LIN {X 0,Y 475.19,Z 422.26,A -85,B 0,C 180,E1 -7300.869,E2 -7300.869} C_VEL
LIN {X 0,Y 475.479,Z 413.975,A -85,B 0,C 180,E1 -7301.294,E2 -7301.294} C_VEL
LIN {X 0,Y 475.705,Z 405.069,A -85,B 0,C 180,E1 -7301.64,E2 -7301.64} C_VEL
LIN {X 0,Y 475.915,Z 396.208,A -85,B 0,C 180,E1 -7301.877,E2 -7301.877} C_VEL
LIN {X 0,Y 476.151,Z 333.395,A -85,B 0,C 180,E1 -7302.878,E2 -7302.878} C_VEL
LIN {X 0,Y 474.49,Z 318.296,A -85,B 0,C 180,E1 -7303.182,E2 -7303.182} C_VEL
LIN {X 0,Y 474.879,Z 302.969,A -85,B 0,C 180,E1 -7305.982,E2 -7305.982} C_VEL
LIN {X 0,Y 475.373,Z 286.697,A -85,B 0,C 180,E1 -7308.981,E2 -7308.981} C_VEL
LIN {X 0,Y 476.015,Z 268.666,A -85,B 0,C 180,E1 -7312.345,E2 -7312.345} C_VEL
LIN {X 0,Y 476.027,Z 263.851,A -85,B 0,C 180,E1 -7313.262,E2 -7313.262} C_VEL
LIN {X 0,Y 474.659,Z 256.174,A -85,B 0,C 180,E1 -7314.843,E2 -7314.843} C_VEL
LIN {X 0,Y 474.641,Z 256.171,A -85,B 0,C 180,E1 -7318.282,E2 -7318.282} C_VEL
LIN {X 0,Y 474.599,Z 256.179,A -85,B 0,C 180,E1 -7321.217,E2 -7321.217} C_VEL
LIN {X 0,Y 474.632,Z 256.171,A -85,B 0,C 180,E1 -7324.241,E2 -7324.241} C_VEL
LIN {X 0,Y 474.589,Z 256.182,A -85,B 0,C 180,E1 -7327.383,E2 -7327.383} C_VEL
LIN {X 0,Y 474.626,Z 256.178,A -85,B 0,C 180,E1 -7329.647,E2 -7329.647} C_VEL
LIN {X 0,Y 474.614,Z 256.174,A -85,B 0,C 180,E1 -7332.934,E2 -7332.934} C_VEL
LIN {X 0,Y 474.606,Z 256.177,A -85,B 0,C 180,E1 -7335.894,E2 -7335.894} C_VEL
LIN {X 0,Y 474.626,Z 256.173,A -85,B 0,C 180,E1 -7339.04,E2 -7339.04} C_VEL
LIN {X 0,Y 474.608,Z 256.18,A -85,B 0,C 180,E1 -7341.703,E2 -7341.703} C_VEL
LIN {X 0,Y 474.626,Z 256.172,A -85,B 0,C 180,E1 -7344.725,E2 -7344.725} C_VEL
LIN {X 0,Y 474.632,Z 256.176,A -85,B 0,C 180,E1 -7347.787,E2 -7347.787} C_VEL
LIN {X 0,Y 474.62,Z 256.173,A -85,B 0,C 180,E1 -7350.884,E2 -7350.884} C_VEL
LIN {X 0,Y 474.664,Z 256.174,A -85,B 0,C 180,E1 -7353.628,E2 -7353.628} C_VEL
LIN {X 0,Y 474.632,Z 256.171,A -85,B 0,C 180,E1 -7356.64,E2 -7356.64} C_VEL
LIN {X 0,Y 474.65,Z 256.17,A -85,B 0,C 180,E1 -7360.089,E2 -7360.089} C_VEL
LIN {X 0,Y 474.645,Z 256.169,A -85,B 0,C 180,E1 -7362.774,E2 -7362.774} C_VEL
LIN {X 0,Y 474.643,Z 256.176,A -85,B 0,C 180,E1 -7365.42,E2 -7365.42} C_VEL
LIN {X 0,Y 474.698,Z 256.165,A -85,B 0,C 180,E1 -7368.037,E2 -7368.037} C_VEL
LIN {X 0,Y 474.723,Z 256.167,A -85,B 0,C 180,E1 -7371.486,E2 -7371.486} C_VEL
LIN {X 0,Y 474.773,Z 256.155,A -85,B 0,C 180,E1 -7374.052,E2 -7374.052} C_VEL
LIN {X 0,Y 474.888,Z 256.145,A -85,B 0,C 180,E1 -7377.455,E2 -7377.455} C_VEL
LIN {X 0,Y 474.905,Z 256.139,A -85,B 0,C 180,E1 -7379.999,E2 -7379.999} C_VEL
LIN {X 0,Y 474.888,Z 256.139,A -85,B 0,C 180,E1 -7382.544,E2 -7382.544} C_VEL
LIN {X 0,Y 474.772,Z 256.157,A -85,B 0,C 180,E1 -7385.947,E2 -7385.947} C_VEL
LIN {X 0,Y 474.721,Z 256.16,A -85,B 0,C 180,E1 -7388.513,E2 -7388.513} C_VEL
LIN {X 0,Y 474.731,Z 256.162,A -85,B 0,C 180,E1 -7391.961,E2 -7391.961} C_VEL
LIN {X 0,Y 474.672,Z 256.171,A -85,B 0,C 180,E1 -7395.767,E2 -7395.767} C_VEL
LIN {X 0,Y 474.657,Z 256.169,A -85,B 0,C 180,E1 -7399.01,E2 -7399.01} C_VEL
LIN {X 0,Y 474.581,Z 256.183,A -85,B 0,C 180,E1 -7401.728,E2 -7401.728} C_VEL
LIN {X 0,Y 474.65,Z 256.169,A -85,B 0,C 180,E1 -7404.492,E2 -7404.492} C_VEL
LIN {X 0,Y 474.69,Z 256.168,A -85,B 0,C 180,E1 -7407.338,E2 -7407.338} C_VEL
LIN {X 0,Y 474.596,Z 256.176,A -85,B 0,C 180,E1 -7410.81,E2 -7410.81} C_VEL
LIN {X 0,Y 474.629,Z 256.174,A -85,B 0,C 180,E1 -7413.984,E2 -7413.984} C_VEL
LIN {X 0,Y 474.566,Z 256.18,A -85,B 0,C 180,E1 -7416.9,E2 -7416.9} C_VEL
LIN {X 0,Y 474.643,Z 256.177,A -85,B 0,C 180,E1 -7419.651,E2 -7419.651} C_VEL
LIN {X 0,Y 474.626,Z 256.173,A -85,B 0,C 180,E1 -7422.931,E2 -7422.931} C_VEL
LIN {X 0,Y 474.609,Z 256.178,A -85,B 0,C 180,E1 -7425.896,E2 -7425.896} C_VEL
LIN {X 0,Y 474.636,Z 256.172,A -85,B 0,C 180,E1 -7429.038,E2 -7429.038} C_VEL
LIN {X 0,Y 474.607,Z 256.181,A -85,B 0,C 180,E1 -7431.703,E2 -7431.703} C_VEL
LIN {X 0,Y 474.619,Z 256.173,A -85,B 0,C 180,E1 -7434.726,E2 -7434.726} C_VEL
LIN {X 0,Y 474.628,Z 256.177,A -85,B 0,C 180,E1 -7437.788,E2 -7437.788} C_VEL
LIN {X 0,Y 474.614,Z 256.174,A -85,B 0,C 180,E1 -7440.884,E2 -7440.884} C_VEL
LIN {X 0,Y 474.652,Z 256.177,A -85,B 0,C 180,E1 -7443.628,E2 -7443.628} C_VEL
LIN {X 0,Y 474.627,Z 256.172,A -85,B 0,C 180,E1 -7446.641,E2 -7446.641} C_VEL
LIN {X 0,Y 474.648,Z 256.171,A -85,B 0,C 180,E1 -7450.089,E2 -7450.089} C_VEL
LIN {X 0,Y 474.646,Z 256.173,A -85,B 0,C 180,E1 -7451.682,E2 -7451.682} C_VEL
LIN {X 0,Y 473.984,Z 256.257,A -85,B 0,C 180,E1 -7452.391,E2 -7452.391} C_VEL
LIN {X 0,Y 471.132,Z 256.614,A -85,B 0,C 180,E1 -7453.542,E2 -7453.542} C_VEL
LIN {X 0,Y 468.716,Z 256.913,A -85,B 0,C 180,E1 -7454.47,E2 -7454.47} C_VEL
LIN {X 0,Y 467.674,Z 257.041,A -85,B 0,C 180,E1 -7455.188,E2 -7455.188} C_VEL
LIN {X 0,Y 467.587,Z 257.05,A -85,B 0,C 180,E1 -7455.431,E2 -7455.431} C_VEL
LIN {X 0,Y 467.646,Z 257.042,A -85,B 0,C 180,E1 -7458.734,E2 -7458.734} C_VEL
LIN {X 0,Y 467.74,Z 257.031,A -85,B 0,C 180,E1 -7462.228,E2 -7462.228} C_VEL
LIN {X 0,Y 467.711,Z 257.034,A -85,B 0,C 180,E1 -7464.827,E2 -7464.827} C_VEL
LIN {X 0,Y 467.849,Z 257.021,A -85,B 0,C 180,E1 -7467.417,E2 -7467.417} C_VEL
LIN {X 0,Y 467.871,Z 257.017,A -85,B 0,C 180,E1 -7470,E2 -7470} C_VEL
LIN {X 0,Y 467.849,Z 257.017,A -85,B 0,C 180,E1 -7472.583,E2 -7472.583} C_VEL
LIN {X 0,Y 467.722,Z 257.035,A -85,B 0,C 180,E1 -7476.037,E2 -7476.037} C_VEL
LIN {X 0,Y 467.671,Z 257.039,A -85,B 0,C 180,E1 -7478.643,E2 -7478.643} C_VEL
LIN {X 0,Y 467.673,Z 257.04,A -85,B 0,C 180,E1 -7482.145,E2 -7482.145} C_VEL
LIN {X 0,Y 467.639,Z 257.047,A -85,B 0,C 180,E1 -7485.885,E2 -7485.885} C_VEL
LIN {X 0,Y 467.612,Z 257.049,A -85,B 0,C 180,E1 -7489.308,E2 -7489.308} C_VEL
LIN {X 0,Y 467.523,Z 257.06,A -85,B 0,C 180,E1 -7492.074,E2 -7492.074} C_VEL
LIN {X 0,Y 467.567,Z 257.053,A -85,B 0,C 180,E1 -7494.889,E2 -7494.889} C_VEL
LIN {X 0,Y 467.604,Z 257.053,A -85,B 0,C 180,E1 -7497.769,E2 -7497.769} C_VEL
LIN {X 0,Y 467.536,Z 257.057,A -85,B 0,C 180,E1 -7501.041,E2 -7501.041} C_VEL
LIN {X 0,Y 467.613,Z 257.233,A -85,B 0,C 180,E1 -7502.883,E2 -7502.883} C_VEL
LIN {X 0,Y 467.517,Z 268.713,A -85,B 0,C 180,E1 -7505.711,E2 -7505.711} C_VEL
LIN {X 0,Y 469.565,Z 280.34,A -85,B 0,C 180,E1 -7505.973,E2 -7505.973} C_VEL
LIN {X 0,Y 469.055,Z 344.667,A -85,B 0,C 180,E1 -7507.011,E2 -7507.011} C_VEL
LIN {X 0,Y 468.902,Z 354.626,A -85,B 0,C 180,E1 -7507.29,E2 -7507.29} C_VEL
LIN {X 0,Y 468.743,Z 365.834,A -85,B 0,C 180,E1 -7507.764,E2 -7507.764} C_VEL
LIN {X 0,Y 468.444,Z 375.752,A -85,B 0,C 180,E1 -7508.357,E2 -7508.357} C_VEL
LIN {X 0,Y 468.184,Z 385.112,A -85,B 0,C 180,E1 -7509.084,E2 -7509.084} C_VEL
LIN {X 0,Y 467.91,Z 392.862,A -85,B 0,C 180,E1 -7509.83,E2 -7509.83} C_VEL
LIN {X 0,Y 467.618,Z 400.12,A -85,B 0,C 180,E1 -7510.684,E2 -7510.684} C_VEL
LIN {X 0,Y 467.375,Z 407.099,A -85,B 0,C 180,E1 -7511.691,E2 -7511.691} C_VEL
LIN {X 0,Y 467.151,Z 413.62,A -85,B 0,C 180,E1 -7512.888,E2 -7512.888} C_VEL
LIN {X 0,Y 466.987,Z 418.643,A -85,B 0,C 180,E1 -7514.098,E2 -7514.098} C_VEL
LIN {X 0,Y 466.865,Z 421.688,A -85,B 0,C 180,E1 -7515.032,E2 -7515.032} C_VEL
LIN {X 0,Y 466.759,Z 424.644,A -85,B 0,C 180,E1 -7516.279,E2 -7516.279} C_VEL
LIN {X 0,Y 466.656,Z 426.538,A -85,B 0,C 180,E1 -7517.556,E2 -7517.556} C_VEL
LIN {X 0,Y 466.634,Z 427.345,A -85,B 0,C 180,E1 -7518.854,E2 -7518.854} C_VEL
LIN {X 0,Y 466.617,Z 426.997,A -85,B 0,C 180,E1 -7520.186,E2 -7520.186} C_VEL
LIN {X 0,Y 466.747,Z 424.688,A -85,B 0,C 180,E1 -7521.878,E2 -7521.878} C_VEL
LIN {X 0,Y 466.892,Z 422.133,A -85,B 0,C 180,E1 -7522.98,E2 -7522.98} C_VEL
LIN {X 0,Y 467.045,Z 417.704,A -85,B 0,C 180,E1 -7524.347,E2 -7524.347} C_VEL
LIN {X 0,Y 467.258,Z 412.531,A -85,B 0,C 180,E1 -7525.507,E2 -7525.507} C_VEL
LIN {X 0,Y 467.451,Z 407.21,A -85,B 0,C 180,E1 -7526.461,E2 -7526.461} C_VEL
LIN {X 0,Y 467.698,Z 399.703,A -85,B 0,C 180,E1 -7527.537,E2 -7527.537} C_VEL
LIN {X 0,Y 468.021,Z 393.235,A -85,B 0,C 180,E1 -7528.294,E2 -7528.294} C_VEL
LIN {X 0,Y 468.283,Z 385.422,A -85,B 0,C 180,E1 -7529.052,E2 -7529.052} C_VEL
LIN {X 0,Y 468.555,Z 376.993,A -85,B 0,C 180,E1 -7529.713,E2 -7529.713} C_VEL
LIN {X 0,Y 468.813,Z 365.724,A -85,B 0,C 180,E1 -7530.396,E2 -7530.396} C_VEL
LIN {X 0,Y 469.014,Z 354.621,A -85,B 0,C 180,E1 -7530.858,E2 -7530.858} C_VEL
LIN {X 0,Y 469.141,Z 345.648,A -85,B 0,C 180,E1 -7531.112,E2 -7531.112} C_VEL
LIN {X 0,Y 469.662,Z 279.9,A -85,B 0,C 180,E1 -7532.183,E2 -7532.183} C_VEL
LIN {X 0,Y 467.626,Z 268.438,A -85,B 0,C 180,E1 -7532.461,E2 -7532.461} C_VEL
LIN {X 0,Y 467.522,Z 257.064,A -85,B 0,C 180,E1 -7534.853,E2 -7534.853} C_VEL
LIN {X 0,Y 467.559,Z 257.059,A -85,B 0,C 180,E1 -7536.996,E2 -7536.996} C_VEL
LIN {X 0,Y 467.612,Z 257.051,A -85,B 0,C 180,E1 -7539.778,E2 -7539.778} C_VEL
LIN {X 0,Y 467.598,Z 257.056,A -85,B 0,C 180,E1 -7542.507,E2 -7542.507} C_VEL
LIN {X 0,Y 467.595,Z 257.05,A -85,B 0,C 180,E1 -7545.197,E2 -7545.197} C_VEL
LIN {X 0,Y 467.646,Z 257.043,A -85,B 0,C 180,E1 -7547.855,E2 -7547.855} C_VEL
LIN {X 0,Y 467.672,Z 257.04,A -85,B 0,C 180,E1 -7551.358,E2 -7551.358} C_VEL
LIN {X 0,Y 467.737,Z 257.033,A -85,B 0,C 180,E1 -7553.963,E2 -7553.963} C_VEL
LIN {X 0,Y 467.851,Z 257.014,A -85,B 0,C 180,E1 -7557.418,E2 -7557.418} C_VEL
LIN {X 0,Y 467.872,Z 257.016,A -85,B 0,C 180,E1 -7560.001,E2 -7560.001} C_VEL
LIN {X 0,Y 467.851,Z 257.023,A -85,B 0,C 180,E1 -7562.584,E2 -7562.584} C_VEL
LIN {X 0,Y 467.735,Z 257.032,A -85,B 0,C 180,E1 -7566.038,E2 -7566.038} C_VEL
LIN {X 0,Y 467.673,Z 257.042,A -85,B 0,C 180,E1 -7568.644,E2 -7568.644} C_VEL
LIN {X 0,Y 467.647,Z 257.044,A -85,B 0,C 180,E1 -7572.146,E2 -7572.146} C_VEL
LIN {X 0,Y 467.631,Z 257.043,A -85,B 0,C 180,E1 -7575.696,E2 -7575.696} C_VEL
LIN {X 0,Y 467.61,Z 257.05,A -85,B 0,C 180,E1 -7578.766,E2 -7578.766} C_VEL
LIN {X 0,Y 467.573,Z 257.047,A -85,B 0,C 180,E1 -7581.269,E2 -7581.269} C_VEL
LIN {X 0,Y 467.566,Z 257.052,A -85,B 0,C 180,E1 -7583.944,E2 -7583.944} C_VEL
LIN {X 0,Y 467.622,Z 257.049,A -85,B 0,C 180,E1 -7586.8,E2 -7586.8} C_VEL
LIN {X 0,Y 467.581,Z 257.045,A -85,B 0,C 180,E1 -7589.737,E2 -7589.737} C_VEL
LIN {X 0,Y 467.578,Z 257.05,A -85,B 0,C 180,E1 -7592.759,E2 -7592.759} C_VEL
LIN {X 0,Y 467.552,Z 257.055,A -85,B 0,C 180,E1 -7595.89,E2 -7595.89} C_VEL
LIN {X 0,Y 467.61,Z 257.047,A -85,B 0,C 180,E1 -7599.142,E2 -7599.142} C_VEL
LIN {X 0,Y 467.582,Z 257.056,A -85,B 0,C 180,E1 -7602.568,E2 -7602.568} C_VEL
LIN {X 0,Y 467.566,Z 257.054,A -85,B 0,C 180,E1 -7605.054,E2 -7605.054} C_VEL
LIN {X 0,Y 467.586,Z 257.049,A -85,B 0,C 180,E1 -7607.441,E2 -7607.441} C_VEL
LIN {X 0,Y 467.579,Z 257.054,A -85,B 0,C 180,E1 -7610.856,E2 -7610.856} C_VEL
LIN {X 0,Y 467.56,Z 257.058,A -85,B 0,C 180,E1 -7614.261,E2 -7614.261} C_VEL
LIN {X 0,Y 467.58,Z 257.051,A -85,B 0,C 180,E1 -7617.322,E2 -7617.322} C_VEL
LIN {X 0,Y 467.567,Z 257.06,A -85,B 0,C 180,E1 -7620.669,E2 -7620.669} C_VEL
LIN {X 0,Y 467.611,Z 257.049,A -85,B 0,C 180,E1 -7623.2,E2 -7623.2} C_VEL
LIN {X 0,Y 467.641,Z 257.128,A -85,B 0,C 180,E1 -7625.648,E2 -7625.648} C_VEL
LIN {X 0,Y 468.758,Z 264.468,A -85,B 0,C 180,E1 -7627.058,E2 -7627.058} C_VEL
LIN {X 0,Y 468.382,Z 277.023,A -85,B 0,C 180,E1 -7629.353,E2 -7629.353} C_VEL
LIN {X 0,Y 467.915,Z 294.514,A -85,B 0,C 180,E1 -7632.519,E2 -7632.519} C_VEL
LIN {X 0,Y 467.473,Z 314.296,A -85,B 0,C 180,E1 -7636.082,E2 -7636.082} C_VEL
LIN {X 0,Y 467.397,Z 317.179,A -85,B 0,C 180,E1 -7636.592,E2 -7636.592} C_VEL
LIN {X 0,Y 469.438,Z 337,A -85,B 0,C 180,E1 -7636.974,E2 -7636.974} C_VEL
LIN {X 0,Y 469.007,Z 395.268,A -85,B 0,C 180,E1 -7637.918,E2 -7637.918} C_VEL
LIN {X 0,Y 468.757,Z 404.976,A -85,B 0,C 180,E1 -7638.186,E2 -7638.186} C_VEL
LIN {X 0,Y 468.411,Z 416.086,A -85,B 0,C 180,E1 -7638.643,E2 -7638.643} C_VEL
LIN {X 0,Y 468.077,Z 426.991,A -85,B 0,C 180,E1 -7639.292,E2 -7639.292} C_VEL
LIN {X 0,Y 467.789,Z 435.462,A -85,B 0,C 180,E1 -7639.942,E2 -7639.942} C_VEL
LIN {X 0,Y 467.48,Z 443.473,A -85,B 0,C 180,E1 -7640.7,E2 -7640.7} C_VEL
LIN {X 0,Y 467.218,Z 450.966,A -85,B 0,C 180,E1 -7641.567,E2 -7641.567} C_VEL
LIN {X 0,Y 467.042,Z 458.58,A -85,B 0,C 180,E1 -7642.652,E2 -7642.652} C_VEL
LIN {X 0,Y 466.811,Z 465.545,A -85,B 0,C 180,E1 -7643.951,E2 -7643.951} C_VEL
LIN {X 0,Y 466.796,Z 469.281,A -85,B 0,C 180,E1 -7644.817,E2 -7644.817} C_VEL
LIN {X 0,Y 466.686,Z 472.339,A -85,B 0,C 180,E1 -7645.682,E2 -7645.682} C_VEL
LIN {X 0,Y 466.762,Z 474.725,A -85,B 0,C 180,E1 -7646.547,E2 -7646.547} C_VEL
LIN {X 0,Y 466.706,Z 476.52,A -85,B 0,C 180,E1 -7647.411,E2 -7647.411} C_VEL
LIN {X 0,Y 466.693,Z 477.808,A -85,B 0,C 180,E1 -7648.274,E2 -7648.274} C_VEL
LIN {X 0,Y 466.626,Z 478.608,A -85,B 0,C 180,E1 -7649.137,E2 -7649.137} C_VEL
LIN {X 0,Y 466.612,Z 478.919,A -85,B 0,C 180,E1 -7650,E2 -7650} C_VEL
LIN {X 0,Y 466.626,Z 478.632,A -85,B 0,C 180,E1 -7650.863,E2 -7650.863} C_VEL
LIN {X 0,Y 466.693,Z 477.841,A -85,B 0,C 180,E1 -7651.726,E2 -7651.726} C_VEL
LIN {X 0,Y 466.706,Z 476.562,A -85,B 0,C 180,E1 -7652.589,E2 -7652.589} C_VEL
LIN {X 0,Y 466.733,Z 473.612,A -85,B 0,C 180,E1 -7653.885,E2 -7653.885} C_VEL
LIN {X 0,Y 466.722,Z 470.906,A -85,B 0,C 180,E1 -7654.751,E2 -7654.751} C_VEL
LIN {X 0,Y 466.817,Z 467.576,A -85,B 0,C 180,E1 -7655.616,E2 -7655.616} C_VEL
LIN {X 0,Y 466.93,Z 462.172,A -85,B 0,C 180,E1 -7656.73,E2 -7656.73} C_VEL
LIN {X 0,Y 467.067,Z 455.786,A -85,B 0,C 180,E1 -7657.783,E2 -7657.783} C_VEL
LIN {X 0,Y 467.385,Z 447.59,A -85,B 0,C 180,E1 -7658.866,E2 -7658.866} C_VEL
LIN {X 0,Y 467.739,Z 437.953,A -85,B 0,C 180,E1 -7659.841,E2 -7659.841} C_VEL
LIN {X 0,Y 467.979,Z 429.95,A -85,B 0,C 180,E1 -7660.492,E2 -7660.492} C_VEL
LIN {X 0,Y 468.214,Z 421.697,A -85,B 0,C 180,E1 -7661.033,E2 -7661.033} C_VEL
LIN {X 0,Y 468.492,Z 413.353,A -85,B 0,C 180,E1 -7661.465,E2 -7661.465} C_VEL
LIN {X 0,Y 468.773,Z 404.358,A -85,B 0,C 180,E1 -7661.814,E2 -7661.814} C_VEL
LIN {X 0,Y 468.94,Z 395.308,A -85,B 0,C 180,E1 -7662.057,E2 -7662.057} C_VEL
LIN {X 0,Y 469.252,Z 334.358,A -85,B 0,C 180,E1 -7663.041,E2 -7663.041} C_VEL
LIN {X 0,Y 467.423,Z 318.062,A -85,B 0,C 180,E1 -7663.355,E2 -7663.355} C_VEL
LIN {X 0,Y 467.868,Z 302.732,A -85,B 0,C 180,E1 -7666.199,E2 -7666.199} C_VEL
LIN {X 0,Y 468.443,Z 285.102,A -85,B 0,C 180,E1 -7669.5,E2 -7669.5} C_VEL
LIN {X 0,Y 469.163,Z 267.094,A -85,B 0,C 180,E1 -7672.922,E2 -7672.922} C_VEL
LIN {X 0,Y 468.122,Z 259.793,A -85,B 0,C 180,E1 -7674.384,E2 -7674.384} C_VEL
LIN {X 0,Y 467.613,Z 257.052,A -85,B 0,C 180,E1 -7674.992,E2 -7674.992} C_VEL
LIN {X 0,Y 467.616,Z 257.051,A -85,B 0,C 180,E1 -7677.769,E2 -7677.769} C_VEL
LIN {X 0,Y 467.568,Z 257.053,A -85,B 0,C 180,E1 -7681.044,E2 -7681.044} C_VEL
LIN {X 0,Y 467.588,Z 257.048,A -85,B 0,C 180,E1 -7684.242,E2 -7684.242} C_VEL
LIN {X 0,Y 467.547,Z 257.057,A -85,B 0,C 180,E1 -7687.186,E2 -7687.186} C_VEL
LIN {X 0,Y 467.576,Z 257.05,A -85,B 0,C 180,E1 -7690.264,E2 -7690.264} C_VEL
LIN {X 0,Y 467.585,Z 257.048,A -85,B 0,C 180,E1 -7692.566,E2 -7692.566} C_VEL
LIN {X 0,Y 467.569,Z 257.053,A -85,B 0,C 180,E1 -7695.052,E2 -7695.052} C_VEL
LIN {X 0,Y 467.587,Z 257.055,A -85,B 0,C 180,E1 -7697.439,E2 -7697.439} C_VEL
LIN {X 0,Y 467.558,Z 257.053,A -85,B 0,C 180,E1 -7700.852,E2 -7700.852} C_VEL
LIN {X 0,Y 467.56,Z 257.052,A -85,B 0,C 180,E1 -7704.26,E2 -7704.26} C_VEL
LIN {X 0,Y 467.579,Z 257.054,A -85,B 0,C 180,E1 -7707.32,E2 -7707.32} C_VEL
LIN {X 0,Y 467.566,Z 257.051,A -85,B 0,C 180,E1 -7710.667,E2 -7710.667} C_VEL
LIN {X 0,Y 467.625,Z 257.047,A -85,B 0,C 180,E1 -7713.2,E2 -7713.2} C_VEL
LIN {X 0,Y 467.589,Z 257.048,A -85,B 0,C 180,E1 -7716.467,E2 -7716.467} C_VEL
LIN {X 0,Y 467.618,Z 257.05,A -85,B 0,C 180,E1 -7719.776,E2 -7719.776} C_VEL
LIN {X 0,Y 467.604,Z 257.046,A -85,B 0,C 180,E1 -7722.506,E2 -7722.506} C_VEL
LIN {X 0,Y 467.601,Z 257.05,A -85,B 0,C 180,E1 -7725.196,E2 -7725.196} C_VEL
LIN {X 0,Y 467.65,Z 257.045,A -85,B 0,C 180,E1 -7727.854,E2 -7727.854} C_VEL
LIN {X 0,Y 467.676,Z 257.042,A -85,B 0,C 180,E1 -7731.357,E2 -7731.357} C_VEL
LIN {X 0,Y 467.737,Z 257.033,A -85,B 0,C 180,E1 -7733.962,E2 -7733.962} C_VEL
LIN {X 0,Y 467.853,Z 257.021,A -85,B 0,C 180,E1 -7737.416,E2 -7737.416} C_VEL
LIN {X 0,Y 467.876,Z 257.015,A -85,B 0,C 180,E1 -7739.999,E2 -7739.999} C_VEL
LIN {X 0,Y 467.854,Z 257.015,A -85,B 0,C 180,E1 -7742.582,E2 -7742.582} C_VEL
LIN {X 0,Y 467.736,Z 257.032,A -85,B 0,C 180,E1 -7746.037,E2 -7746.037} C_VEL
LIN {X 0,Y 467.674,Z 257.038,A -85,B 0,C 180,E1 -7748.642,E2 -7748.642} C_VEL
LIN {X 0,Y 467.675,Z 257.039,A -85,B 0,C 180,E1 -7752.144,E2 -7752.144} C_VEL
LIN {X 0,Y 467.641,Z 257.046,A -85,B 0,C 180,E1 -7755.885,E2 -7755.885} C_VEL
LIN {X 0,Y 467.616,Z 257.049,A -85,B 0,C 180,E1 -7759.307,E2 -7759.307} C_VEL
LIN {X 0,Y 467.526,Z 257.058,A -85,B 0,C 180,E1 -7762.073,E2 -7762.073} C_VEL
LIN {X 0,Y 467.595,Z 257.049,A -85,B 0,C 180,E1 -7764.887,E2 -7764.887} C_VEL
LIN {X 0,Y 467.618,Z 257.05,A -85,B 0,C 180,E1 -7767.768,E2 -7767.768} C_VEL
LIN {X 0,Y 467.56,Z 257.054,A -85,B 0,C 180,E1 -7771.045,E2 -7771.045} C_VEL
LIN {X 0,Y 467.581,Z 257.05,A -85,B 0,C 180,E1 -7774.242,E2 -7774.242} C_VEL
LIN {X 0,Y 467.542,Z 257.057,A -85,B 0,C 180,E1 -7777.187,E2 -7777.187} C_VEL
LIN {X 0,Y 467.587,Z 257.05,A -85,B 0,C 180,E1 -7780.262,E2 -7780.262} C_VEL
LIN {X 0,Y 467.577,Z 257.05,A -85,B 0,C 180,E1 -7782.567,E2 -7782.567} C_VEL
LIN {X 0,Y 467.561,Z 257.054,A -85,B 0,C 180,E1 -7785.053,E2 -7785.053} C_VEL
LIN {X 0,Y 467.615,Z 257.051,A -85,B 0,C 180,E1 -7787.444,E2 -7787.444} C_VEL
LIN {X 0,Y 467.59,Z 257.049,A -85,B 0,C 180,E1 -7790.857,E2 -7790.857} C_VEL
LIN {X 0,Y 467.553,Z 257.054,A -85,B 0,C 180,E1 -7794.26,E2 -7794.26} C_VEL
LIN {X 0,Y 467.573,Z 257.054,A -85,B 0,C 180,E1 -7797.32,E2 -7797.32} C_VEL
LIN {X 0,Y 467.56,Z 257.052,A -85,B 0,C 180,E1 -7800.667,E2 -7800.667} C_VEL
LIN {X 0,Y 467.607,Z 257.049,A -85,B 0,C 180,E1 -7803.2,E2 -7803.2} C_VEL
LIN {X 0,Y 467.585,Z 257.049,A -85,B 0,C 180,E1 -7806.468,E2 -7806.468} C_VEL
LIN {X 0,Y 467.615,Z 257.051,A -85,B 0,C 180,E1 -7809.777,E2 -7809.777} C_VEL
LIN {X 0,Y 467.6,Z 257.047,A -85,B 0,C 180,E1 -7812.507,E2 -7812.507} C_VEL
LIN {X 0,Y 467.587,Z 257.05,A -85,B 0,C 180,E1 -7815.431,E2 -7815.431} C_VEL
LIN {X 0,Y 466.918,Z 257.135,A -85,B 0,C 180,E1 -7816.15,E2 -7816.15} C_VEL
LIN {X 0,Y 464.075,Z 257.49,A -85,B 0,C 180,E1 -7817.318,E2 -7817.318} C_VEL
LIN {X 0,Y 461.677,Z 257.786,A -85,B 0,C 180,E1 -7818.26,E2 -7818.26} C_VEL
LIN {X 0,Y 460.652,Z 257.914,A -85,B 0,C 180,E1 -7818.988,E2 -7818.988} C_VEL
LIN {X 0,Y 460.57,Z 257.925,A -85,B 0,C 180,E1 -7819.234,E2 -7819.234} C_VEL
LIN {X 0,Y 460.706,Z 257.906,A -85,B 0,C 180,E1 -7822.543,E2 -7822.543} C_VEL
LIN {X 0,Y 460.684,Z 257.909,A -85,B 0,C 180,E1 -7824.748,E2 -7824.748} C_VEL
LIN {X 0,Y 460.79,Z 257.9,A -85,B 0,C 180,E1 -7827.377,E2 -7827.377} C_VEL
LIN {X 0,Y 460.842,Z 257.892,A -85,B 0,C 180,E1 -7830,E2 -7830} C_VEL
LIN {X 0,Y 460.79,Z 257.896,A -85,B 0,C 180,E1 -7832.622,E2 -7832.622} C_VEL
LIN {X 0,Y 460.688,Z 257.91,A -85,B 0,C 180,E1 -7836.13,E2 -7836.13} C_VEL
LIN {X 0,Y 460.618,Z 257.918,A -85,B 0,C 180,E1 -7838.776,E2 -7838.776} C_VEL
LIN {X 0,Y 460.624,Z 257.917,A -85,B 0,C 180,E1 -7842.457,E2 -7842.457} C_VEL
LIN {X 0,Y 460.59,Z 257.924,A -85,B 0,C 180,E1 -7845.997,E2 -7845.997} C_VEL
LIN {X 0,Y 460.559,Z 257.926,A -85,B 0,C 180,E1 -7848.901,E2 -7848.901} C_VEL
LIN {X 0,Y 460.505,Z 257.936,A -85,B 0,C 180,E1 -7851.485,E2 -7851.485} C_VEL
LIN {X 0,Y 460.514,Z 257.931,A -85,B 0,C 180,E1 -7854.333,E2 -7854.333} C_VEL
LIN {X 0,Y 460.566,Z 257.93,A -85,B 0,C 180,E1 -7857.745,E2 -7857.745} C_VEL
LIN {X 0,Y 460.509,Z 257.935,A -85,B 0,C 180,E1 -7861.257,E2 -7861.257} C_VEL
LIN {X 0,Y 460.566,Z 258.083,A -85,B 0,C 180,E1 -7862.799,E2 -7862.799} C_VEL
LIN {X 0,Y 460.508,Z 266.701,A -85,B 0,C 180,E1 -7864.942,E2 -7864.942} C_VEL
LIN {X 0,Y 460.502,Z 269.068,A -85,B 0,C 180,E1 -7865.523,E2 -7865.523} C_VEL
LIN {X 0,Y 462.634,Z 281.728,A -85,B 0,C 180,E1 -7865.802,E2 -7865.802} C_VEL
LIN {X 0,Y 462.115,Z 344.743,A -85,B 0,C 180,E1 -7866.836,E2 -7866.836} C_VEL
LIN {X 0,Y 461.916,Z 354.557,A -85,B 0,C 180,E1 -7867.11,E2 -7867.11} C_VEL
LIN {X 0,Y 461.792,Z 365.886,A -85,B 0,C 180,E1 -7867.59,E2 -7867.59} C_VEL
LIN {X 0,Y 461.491,Z 374.985,A -85,B 0,C 180,E1 -7868.125,E2 -7868.125} C_VEL
LIN {X 0,Y 461.256,Z 384.108,A -85,B 0,C 180,E1 -7868.823,E2 -7868.823} C_VEL
LIN {X 0,Y 460.951,Z 392.262,A -85,B 0,C 180,E1 -7869.599,E2 -7869.599} C_VEL
LIN {X 0,Y 460.635,Z 399.359,A -85,B 0,C 180,E1 -7870.423,E2 -7870.423} C_VEL
LIN {X 0,Y 460.423,Z 405.561,A -85,B 0,C 180,E1 -7871.296,E2 -7871.296} C_VEL
LIN {X 0,Y 460.206,Z 410.973,A -85,B 0,C 180,E1 -7872.216,E2 -7872.216} C_VEL
LIN {X 0,Y 459.977,Z 416.757,A -85,B 0,C 180,E1 -7873.436,E2 -7873.436} C_VEL
LIN {X 0,Y 459.844,Z 421.216,A -85,B 0,C 180,E1 -7874.67,E2 -7874.67} C_VEL
LIN {X 0,Y 459.714,Z 424.44,A -85,B 0,C 180,E1 -7875.931,E2 -7875.931} C_VEL
LIN {X 0,Y 459.591,Z 426.566,A -85,B 0,C 180,E1 -7877.222,E2 -7877.222} C_VEL
LIN {X 0,Y 459.545,Z 427.609,A -85,B 0,C 180,E1 -7878.535,E2 -7878.535} C_VEL
LIN {X 0,Y 459.544,Z 427.488,A -85,B 0,C 180,E1 -7880.036,E2 -7880.036} C_VEL
LIN {X 0,Y 459.618,Z 426.287,A -85,B 0,C 180,E1 -7881.244,E2 -7881.244} C_VEL
LIN {X 0,Y 459.783,Z 423.596,A -85,B 0,C 180,E1 -7882.639,E2 -7882.639} C_VEL
LIN {X 0,Y 459.908,Z 420.353,A -85,B 0,C 180,E1 -7883.782,E2 -7883.782} C_VEL
LIN {X 0,Y 460.073,Z 416.641,A -85,B 0,C 180,E1 -7884.785,E2 -7884.785} C_VEL
LIN {X 0,Y 460.272,Z 411.584,A -85,B 0,C 180,E1 -7885.866,E2 -7885.866} C_VEL
LIN {X 0,Y 460.444,Z 407.035,A -85,B 0,C 180,E1 -7886.669,E2 -7886.669} C_VEL
LIN {X 0,Y 460.666,Z 400.932,A -85,B 0,C 180,E1 -7887.565,E2 -7887.565} C_VEL
LIN {X 0,Y 461.032,Z 393.607,A -85,B 0,C 180,E1 -7888.443,E2 -7888.443} C_VEL
LIN {X 0,Y 461.309,Z 386.075,A -85,B 0,C 180,E1 -7889.186,E2 -7889.186} C_VEL
LIN {X 0,Y 461.596,Z 377.93,A -85,B 0,C 180,E1 -7889.84,E2 -7889.84} C_VEL
LIN {X 0,Y 461.798,Z 368.787,A -85,B 0,C 180,E1 -7890.425,E2 -7890.425} C_VEL
LIN {X 0,Y 462.064,Z 356.373,A -85,B 0,C 180,E1 -7890.996,E2 -7890.996} C_VEL
LIN {X 0,Y 462.219,Z 346.142,A -85,B 0,C 180,E1 -7891.297,E2 -7891.297} C_VEL
LIN {X 0,Y 462.712,Z 280.086,A -85,B 0,C 180,E1 -7892.401,E2 -7892.401} C_VEL
LIN {X 0,Y 460.64,Z 268.889,A -85,B 0,C 180,E1 -7892.666,E2 -7892.666} C_VEL
LIN {X 0,Y 460.634,Z 259.161,A -85,B 0,C 180,E1 -7894.711,E2 -7894.711} C_VEL
LIN {X 0,Y 460.488,Z 257.939,A -85,B 0,C 180,E1 -7895.004,E2 -7895.004} C_VEL
LIN {X 0,Y 460.495,Z 257.937,A -85,B 0,C 180,E1 -7897.572,E2 -7897.572} C_VEL
LIN {X 0,Y 460.558,Z 257.935,A -85,B 0,C 180,E1 -7900.385,E2 -7900.385} C_VEL
LIN {X 0,Y 460.555,Z 257.928,A -85,B 0,C 180,E1 -7903.147,E2 -7903.147} C_VEL
LIN {X 0,Y 460.543,Z 257.929,A -85,B 0,C 180,E1 -7905.868,E2 -7905.868} C_VEL
LIN {X 0,Y 460.603,Z 257.927,A -85,B 0,C 180,E1 -7908.56,E2 -7908.56} C_VEL
LIN {X 0,Y 460.685,Z 257.913,A -85,B 0,C 180,E1 -7912.109,E2 -7912.109} C_VEL
LIN {X 0,Y 460.692,Z 257.912,A -85,B 0,C 180,E1 -7914.749,E2 -7914.749} C_VEL
LIN {X 0,Y 460.816,Z 257.891,A -85,B 0,C 180,E1 -7917.378,E2 -7917.378} C_VEL
LIN {X 0,Y 460.843,Z 257.892,A -85,B 0,C 180,E1 -7920.001,E2 -7920.001} C_VEL
LIN {X 0,Y 460.816,Z 257.898,A -85,B 0,C 180,E1 -7922.623,E2 -7922.623} C_VEL
LIN {X 0,Y 460.701,Z 257.909,A -85,B 0,C 180,E1 -7926.131,E2 -7926.131} C_VEL
LIN {X 0,Y 460.62,Z 257.92,A -85,B 0,C 180,E1 -7928.777,E2 -7928.777} C_VEL
LIN {X 0,Y 460.605,Z 257.921,A -85,B 0,C 180,E1 -7932.446,E2 -7932.446} C_VEL
LIN {X 0,Y 460.592,Z 257.921,A -85,B 0,C 180,E1 -7935.998,E2 -7935.998} C_VEL
LIN {X 0,Y 460.563,Z 257.926,A -85,B 0,C 180,E1 -7938.903,E2 -7938.903} C_VEL
LIN {X 0,Y 460.509,Z 257.927,A -85,B 0,C 180,E1 -7941.487,E2 -7941.487} C_VEL
LIN {X 0,Y 460.536,Z 257.932,A -85,B 0,C 180,E1 -7944.333,E2 -7944.333} C_VEL
LIN {X 0,Y 460.578,Z 257.922,A -85,B 0,C 180,E1 -7947.244,E2 -7947.244} C_VEL
LIN {X 0,Y 460.521,Z 257.929,A -85,B 0,C 180,E1 -7950.24,E2 -7950.24} C_VEL
LIN {X 0,Y 460.523,Z 257.924,A -85,B 0,C 180,E1 -7953.326,E2 -7953.326} C_VEL
LIN {X 0,Y 460.474,Z 257.939,A -85,B 0,C 180,E1 -7956.53,E2 -7956.53} C_VEL
LIN {X 0,Y 460.571,Z 257.924,A -85,B 0,C 180,E1 -7959.859,E2 -7959.859} C_VEL
LIN {X 0,Y 460.508,Z 257.932,A -85,B 0,C 180,E1 -7962.901,E2 -7962.901} C_VEL
LIN {X 0,Y 460.508,Z 257.932,A -85,B 0,C 180,E1 -7965.831,E2 -7965.831} C_VEL
LIN {X 0,Y 460.528,Z 257.931,A -85,B 0,C 180,E1 -7968.99,E2 -7968.99} C_VEL
LIN {X 0,Y 460.523,Z 257.93,A -85,B 0,C 180,E1 -7971.268,E2 -7971.268} C_VEL
LIN {X 0,Y 460.51,Z 257.938,A -85,B 0,C 180,E1 -7974.555,E2 -7974.555} C_VEL
LIN {X 0,Y 460.53,Z 257.93,A -85,B 0,C 180,E1 -7977.716,E2 -7977.716} C_VEL
LIN {X 0,Y 460.537,Z 257.935,A -85,B 0,C 180,E1 -7980.77,E2 -7980.77} C_VEL
LIN {X 0,Y 460.555,Z 257.928,A -85,B 0,C 180,E1 -7983.735,E2 -7983.735} C_VEL
LIN {X 0,Y 460.574,Z 257.966,A -85,B 0,C 180,E1 -7985.49,E2 -7985.49} C_VEL
LIN {X 0,Y 461.763,Z 265.308,A -85,B 0,C 180,E1 -7986.927,E2 -7986.927} C_VEL
LIN {X 0,Y 461.382,Z 277.874,A -85,B 0,C 180,E1 -7989.259,E2 -7989.259} C_VEL
LIN {X 0,Y 460.907,Z 294.117,A -85,B 0,C 180,E1 -7992.245,E2 -7992.245} C_VEL
LIN {X 0,Y 460.494,Z 311.467,A -85,B 0,C 180,E1 -7995.415,E2 -7995.415} C_VEL
LIN {X 0,Y 460.377,Z 316.646,A -85,B 0,C 180,E1 -7996.358,E2 -7996.358} C_VEL
LIN {X 0,Y 462.529,Z 336.758,A -85,B 0,C 180,E1 -7996.771,E2 -7996.771} C_VEL
LIN {X 0,Y 462.073,Z 395.041,A -85,B 0,C 180,E1 -7997.734,E2 -7997.734} C_VEL
LIN {X 0,Y 461.797,Z 405.504,A -85,B 0,C 180,E1 -7998.033,E2 -7998.033} C_VEL
LIN {X 0,Y 461.375,Z 417.756,A -85,B 0,C 180,E1 -7998.579,E2 -7998.579} C_VEL
LIN {X 0,Y 461.063,Z 426.628,A -85,B 0,C 180,E1 -7999.127,E2 -7999.127} C_VEL
LIN {X 0,Y 460.767,Z 435.092,A -85,B 0,C 180,E1 -7999.787,E2 -7999.787} C_VEL
LIN {X 0,Y 460.463,Z 443.101,A -85,B 0,C 180,E1 -8000.557,E2 -8000.557} C_VEL
LIN {X 0,Y 460.174,Z 450.593,A -85,B 0,C 180,E1 -8001.437,E2 -8001.437} C_VEL
LIN {X 0,Y 459.965,Z 458.204,A -85,B 0,C 180,E1 -8002.538,E2 -8002.538} C_VEL
LIN {X 0,Y 459.72,Z 465.163,A -85,B 0,C 180,E1 -8003.857,E2 -8003.857} C_VEL
LIN {X 0,Y 459.652,Z 470.449,A -85,B 0,C 180,E1 -8005.176,E2 -8005.176} C_VEL
LIN {X 0,Y 459.66,Z 474.345,A -85,B 0,C 180,E1 -8006.494,E2 -8006.494} C_VEL
LIN {X 0,Y 459.627,Z 476.135,A -85,B 0,C 180,E1 -8007.371,E2 -8007.371} C_VEL
LIN {X 0,Y 459.6,Z 477.419,A -85,B 0,C 180,E1 -8008.248,E2 -8008.248} C_VEL
LIN {X 0,Y 459.559,Z 478.218,A -85,B 0,C 180,E1 -8009.124,E2 -8009.124} C_VEL
LIN {X 0,Y 459.543,Z 478.527,A -85,B 0,C 180,E1 -8010,E2 -8010} C_VEL
LIN {X 0,Y 459.559,Z 478.239,A -85,B 0,C 180,E1 -8010.876,E2 -8010.876} C_VEL
LIN {X 0,Y 459.6,Z 477.441,A -85,B 0,C 180,E1 -8011.753,E2 -8011.753} C_VEL
LIN {X 0,Y 459.627,Z 476.156,A -85,B 0,C 180,E1 -8012.629,E2 -8012.629} C_VEL
LIN {X 0,Y 459.628,Z 473.195,A -85,B 0,C 180,E1 -8013.946,E2 -8013.946} C_VEL
LIN {X 0,Y 459.652,Z 470.48,A -85,B 0,C 180,E1 -8014.824,E2 -8014.824} C_VEL
LIN {X 0,Y 459.714,Z 467.135,A -85,B 0,C 180,E1 -8015.703,E2 -8015.703} C_VEL
LIN {X 0,Y 459.839,Z 462.094,A -85,B 0,C 180,E1 -8016.764,E2 -8016.764} C_VEL
LIN {X 0,Y 459.975,Z 456.74,A -85,B 0,C 180,E1 -8017.683,E2 -8017.683} C_VEL
LIN {X 0,Y 460.183,Z 450.544,A -85,B 0,C 180,E1 -8018.563,E2 -8018.563} C_VEL
LIN {X 0,Y 460.423,Z 444.036,A -85,B 0,C 180,E1 -8019.334,E2 -8019.334} C_VEL
LIN {X 0,Y 460.729,Z 436.158,A -85,B 0,C 180,E1 -8020.103,E2 -8020.103} C_VEL
LIN {X 0,Y 461.056,Z 427.853,A -85,B 0,C 180,E1 -8020.762,E2 -8020.762} C_VEL
LIN {X 0,Y 461.313,Z 419.181,A -85,B 0,C 180,E1 -8021.312,E2 -8021.312} C_VEL
LIN {X 0,Y 461.675,Z 407.627,A -85,B 0,C 180,E1 -8021.859,E2 -8021.859} C_VEL
LIN {X 0,Y 461.984,Z 396.785,A -85,B 0,C 180,E1 -8022.185,E2 -8022.185} C_VEL
LIN {X 0,Y 462.266,Z 368.852,A -85,B 0,C 180,E1 -8022.661,E2 -8022.661} C_VEL
LIN {X 0,Y 462.319,Z 334.854,A -85,B 0,C 180,E1 -8023.214,E2 -8023.214} C_VEL
LIN {X 0,Y 460.415,Z 317.648,A -85,B 0,C 180,E1 -8023.562,E2 -8023.562} C_VEL
LIN {X 0,Y 460.867,Z 301.588,A -85,B 0,C 180,E1 -8026.591,E2 -8026.591} C_VEL
LIN {X 0,Y 461.519,Z 283.513,A -85,B 0,C 180,E1 -8030.037,E2 -8030.037} C_VEL
LIN {X 0,Y 462.178,Z 267.882,A -85,B 0,C 180,E1 -8033.051,E2 -8033.051} C_VEL
LIN {X 0,Y 460.556,Z 257.931,A -85,B 0,C 180,E1 -8035.113,E2 -8035.113} C_VEL
LIN {X 0,Y 460.549,Z 257.927,A -85,B 0,C 180,E1 -8038.233,E2 -8038.233} C_VEL
LIN {X 0,Y 460.521,Z 257.933,A -85,B 0,C 180,E1 -8041.282,E2 -8041.282} C_VEL
LIN {X 0,Y 460.532,Z 257.927,A -85,B 0,C 180,E1 -8044.505,E2 -8044.505} C_VEL
LIN {X 0,Y 460.5,Z 257.938,A -85,B 0,C 180,E1 -8047.623,E2 -8047.623} C_VEL
LIN {X 0,Y 460.541,Z 257.926,A -85,B 0,C 180,E1 -8050.269,E2 -8050.269} C_VEL
LIN {X 0,Y 460.499,Z 257.937,A -85,B 0,C 180,E1 -8053.375,E2 -8053.375} C_VEL
LIN {X 0,Y 460.496,Z 257.932,A -85,B 0,C 180,E1 -8056.624,E2 -8056.624} C_VEL
LIN {X 0,Y 460.537,Z 257.932,A -85,B 0,C 180,E1 -8059.73,E2 -8059.73} C_VEL
LIN {X 0,Y 460.498,Z 257.931,A -85,B 0,C 180,E1 -8062.523,E2 -8062.523} C_VEL
LIN {X 0,Y 460.545,Z 257.933,A -85,B 0,C 180,E1 -8065.623,E2 -8065.623} C_VEL
LIN {X 0,Y 460.534,Z 257.927,A -85,B 0,C 180,E1 -8068.744,E2 -8068.744} C_VEL
LIN {X 0,Y 460.585,Z 257.921,A -85,B 0,C 180,E1 -8072.251,E2 -8072.251} C_VEL
LIN {X 0,Y 460.556,Z 257.924,A -85,B 0,C 180,E1 -8074.705,E2 -8074.705} C_VEL
LIN {X 0,Y 460.508,Z 257.938,A -85,B 0,C 180,E1 -8077.571,E2 -8077.571} C_VEL
LIN {X 0,Y 460.564,Z 257.923,A -85,B 0,C 180,E1 -8080.384,E2 -8080.384} C_VEL
LIN {X 0,Y 460.56,Z 257.926,A -85,B 0,C 180,E1 -8083.145,E2 -8083.145} C_VEL
LIN {X 0,Y 460.55,Z 257.929,A -85,B 0,C 180,E1 -8085.867,E2 -8085.867} C_VEL
LIN {X 0,Y 460.606,Z 257.918,A -85,B 0,C 180,E1 -8088.559,E2 -8088.559} C_VEL
LIN {X 0,Y 460.69,Z 257.909,A -85,B 0,C 180,E1 -8092.108,E2 -8092.108} C_VEL
LIN {X 0,Y 460.692,Z 257.908,A -85,B 0,C 180,E1 -8094.748,E2 -8094.748} C_VEL
LIN {X 0,Y 460.818,Z 257.897,A -85,B 0,C 180,E1 -8097.377,E2 -8097.377} C_VEL
LIN {X 0,Y 460.846,Z 257.891,A -85,B 0,C 180,E1 -8099.999,E2 -8099.999} C_VEL
LIN {X 0,Y 460.819,Z 257.892,A -85,B 0,C 180,E1 -8102.622,E2 -8102.622} C_VEL
LIN {X 0,Y 460.702,Z 257.908,A -85,B 0,C 180,E1 -8106.129,E2 -8106.129} C_VEL
LIN {X 0,Y 460.622,Z 257.917,A -85,B 0,C 180,E1 -8108.775,E2 -8108.775} C_VEL
LIN {X 0,Y 460.627,Z 257.916,A -85,B 0,C 180,E1 -8112.456,E2 -8112.456} C_VEL
LIN {X 0,Y 460.592,Z 257.923,A -85,B 0,C 180,E1 -8115.997,E2 -8115.997} C_VEL
LIN {X 0,Y 460.563,Z 257.925,A -85,B 0,C 180,E1 -8118.901,E2 -8118.901} C_VEL
LIN {X 0,Y 460.507,Z 257.937,A -85,B 0,C 180,E1 -8121.485,E2 -8121.485} C_VEL
LIN {X 0,Y 460.534,Z 257.928,A -85,B 0,C 180,E1 -8124.332,E2 -8124.332} C_VEL
LIN {X 0,Y 460.575,Z 257.925,A -85,B 0,C 180,E1 -8127.243,E2 -8127.243} C_VEL
LIN {X 0,Y 460.502,Z 257.932,A -85,B 0,C 180,E1 -8130.239,E2 -8130.239} C_VEL
LIN {X 0,Y 460.52,Z 257.933,A -85,B 0,C 180,E1 -8133.324,E2 -8133.324} C_VEL
LIN {X 0,Y 460.47,Z 257.935,A -85,B 0,C 180,E1 -8136.529,E2 -8136.529} C_VEL
LIN {X 0,Y 460.567,Z 257.928,A -85,B 0,C 180,E1 -8139.857,E2 -8139.857} C_VEL
LIN {X 0,Y 460.507,Z 257.932,A -85,B 0,C 180,E1 -8142.9,E2 -8142.9} C_VEL
LIN {X 0,Y 460.514,Z 257.935,A -85,B 0,C 180,E1 -8145.828,E2 -8145.828} C_VEL
LIN {X 0,Y 460.533,Z 257.929,A -85,B 0,C 180,E1 -8148.99,E2 -8148.99} C_VEL
LIN {X 0,Y 460.53,Z 257.931,A -85,B 0,C 180,E1 -8151.268,E2 -8151.268} C_VEL
LIN {X 0,Y 460.503,Z 257.931,A -85,B 0,C 180,E1 -8154.554,E2 -8154.554} C_VEL
LIN {X 0,Y 460.523,Z 257.935,A -85,B 0,C 180,E1 -8157.715,E2 -8157.715} C_VEL
LIN {X 0,Y 460.53,Z 257.928,A -85,B 0,C 180,E1 -8160.769,E2 -8160.769} C_VEL
LIN {X 0,Y 460.554,Z 257.931,A -85,B 0,C 180,E1 -8163.735,E2 -8163.735} C_VEL
LIN {X 0,Y 460.538,Z 257.927,A -85,B 0,C 180,E1 -8166.624,E2 -8166.624} C_VEL
LIN {X 0,Y 460.545,Z 257.931,A -85,B 0,C 180,E1 -8169.453,E2 -8169.453} C_VEL
LIN {X 0,Y 460.55,Z 257.927,A -85,B 0,C 180,E1 -8172.23,E2 -8172.23} C_VEL
LIN {X 0,Y 460.556,Z 257.926,A -85,B 0,C 180,E1 -8174.965,E2 -8174.965} C_VEL
LIN {X 0,Y 460.604,Z 257.919,A -85,B 0,C 180,E1 -8178.559,E2 -8178.559} C_VEL
LIN {X 0,Y 460.57,Z 257.925,A -85,B 0,C 180,E1 -8179.234,E2 -8179.234} C_VEL
LIN {X 0,Y 459.915,Z 258.012,A -85,B 0,C 180,E1 -8179.964,E2 -8179.964} C_VEL
LIN {X 0,Y 457.093,Z 258.363,A -85,B 0,C 180,E1 -8181.151,E2 -8181.151} C_VEL
LIN {X 0,Y 454.71,Z 258.656,A -85,B 0,C 180,E1 -8182.108,E2 -8182.108} C_VEL
LIN {X 0,Y 453.696,Z 258.78,A -85,B 0,C 180,E1 -8182.847,E2 -8182.847} C_VEL
LIN {X 0,Y 453.619,Z 258.79,A -85,B 0,C 180,E1 -8183.097,E2 -8183.097} C_VEL
LIN {X 0,Y 453.657,Z 258.785,A -85,B 0,C 180,E1 -8184.666,E2 -8184.666} C_VEL
LIN {X 0,Y 453.734,Z 258.778,A -85,B 0,C 180,E1 -8187.336,E2 -8187.336} C_VEL
LIN {X 0,Y 453.812,Z 258.768,A -85,B 0,C 180,E1 -8190,E2 -8190} C_VEL
LIN {X 0,Y 453.734,Z 258.775,A -85,B 0,C 180,E1 -8192.663,E2 -8192.663} C_VEL
LIN {X 0,Y 453.656,Z 258.786,A -85,B 0,C 180,E1 -8196.225,E2 -8196.225} C_VEL
LIN {X 0,Y 453.582,Z 258.795,A -85,B 0,C 180,E1 -8198.913,E2 -8198.913} C_VEL
LIN {X 0,Y 453.592,Z 258.793,A -85,B 0,C 180,E1 -8202.551,E2 -8202.551} C_VEL
LIN {X 0,Y 453.534,Z 258.801,A -85,B 0,C 180,E1 -8206.196,E2 -8206.196} C_VEL
LIN {X 0,Y 453.509,Z 258.804,A -85,B 0,C 180,E1 -8209.04,E2 -8209.04} C_VEL
LIN {X 0,Y 453.465,Z 258.813,A -85,B 0,C 180,E1 -8211.836,E2 -8211.836} C_VEL
LIN {X 0,Y 453.484,Z 258.806,A -85,B 0,C 180,E1 -8214.735,E2 -8214.735} C_VEL
LIN {X 0,Y 453.517,Z 258.806,A -85,B 0,C 180,E1 -8217.959,E2 -8217.959} C_VEL
LIN {X 0,Y 453.454,Z 258.817,A -85,B 0,C 180,E1 -8221.525,E2 -8221.525} C_VEL
LIN {X 0,Y 453.533,Z 258.961,A -85,B 0,C 180,E1 -8222.712,E2 -8222.712} C_VEL
LIN {X 0,Y 453.512,Z 268.033,A -85,B 0,C 180,E1 -8224.985,E2 -8224.985} C_VEL
LIN {X 0,Y 453.504,Z 269.403,A -85,B 0,C 180,E1 -8225.325,E2 -8225.325} C_VEL
LIN {X 0,Y 455.726,Z 282.642,A -85,B 0,C 180,E1 -8225.619,E2 -8225.619} C_VEL
LIN {X 0,Y 455.171,Z 345.456,A -85,B 0,C 180,E1 -8226.67,E2 -8226.67} C_VEL
LIN {X 0,Y 454.975,Z 355.366,A -85,B 0,C 180,E1 -8226.956,E2 -8226.956} C_VEL
LIN {X 0,Y 454.828,Z 367.119,A -85,B 0,C 180,E1 -8227.474,E2 -8227.474} C_VEL
LIN {X 0,Y 454.511,Z 376.227,A -85,B 0,C 180,E1 -8228.035,E2 -8228.035} C_VEL
LIN {X 0,Y 454.268,Z 384.209,A -85,B 0,C 180,E1 -8228.655,E2 -8228.655} C_VEL
LIN {X 0,Y 453.977,Z 392.004,A -85,B 0,C 180,E1 -8229.398,E2 -8229.398} C_VEL
LIN {X 0,Y 453.61,Z 399.742,A -85,B 0,C 180,E1 -8230.303,E2 -8230.303} C_VEL
LIN {X 0,Y 453.389,Z 406.052,A -85,B 0,C 180,E1 -8231.207,E2 -8231.207} C_VEL
LIN {X 0,Y 453.09,Z 413.034,A -85,B 0,C 180,E1 -8232.44,E2 -8232.44} C_VEL
LIN {X 0,Y 452.875,Z 418.51,A -85,B 0,C 180,E1 -8233.706,E2 -8233.706} C_VEL
LIN {X 0,Y 452.725,Z 422.752,A -85,B 0,C 180,E1 -8235.044,E2 -8235.044} C_VEL
LIN {X 0,Y 452.647,Z 424.398,A -85,B 0,C 180,E1 -8235.68,E2 -8235.68} C_VEL
LIN {X 0,Y 452.526,Z 426.611,A -85,B 0,C 180,E1 -8236.896,E2 -8236.896} C_VEL
LIN {X 0,Y 452.462,Z 427.874,A -85,B 0,C 180,E1 -8238.207,E2 -8238.207} C_VEL
LIN {X 0,Y 452.463,Z 428.048,A -85,B 0,C 180,E1 -8239.56,E2 -8239.56} C_VEL
LIN {X 0,Y 452.503,Z 427.055,A -85,B 0,C 180,E1 -8240.946,E2 -8240.946} C_VEL
LIN {X 0,Y 452.674,Z 424.815,A -85,B 0,C 180,E1 -8242.352,E2 -8242.352} C_VEL
LIN {X 0,Y 452.856,Z 420.748,A -85,B 0,C 180,E1 -8243.863,E2 -8243.863} C_VEL
LIN {X 0,Y 453.062,Z 416.638,A -85,B 0,C 180,E1 -8244.975,E2 -8244.975} C_VEL
LIN {X 0,Y 453.27,Z 411.498,A -85,B 0,C 180,E1 -8246.071,E2 -8246.071} C_VEL
LIN {X 0,Y 453.478,Z 406.223,A -85,B 0,C 180,E1 -8246.986,E2 -8246.986} C_VEL
LIN {X 0,Y 453.725,Z 400.374,A -85,B 0,C 180,E1 -8247.83,E2 -8247.83} C_VEL
LIN {X 0,Y 454.035,Z 394.254,A -85,B 0,C 180,E1 -8248.57,E2 -8248.57} C_VEL
LIN {X 0,Y 454.329,Z 386.974,A -85,B 0,C 180,E1 -8249.306,E2 -8249.306} C_VEL
LIN {X 0,Y 454.625,Z 379.075,A -85,B 0,C 180,E1 -8249.96,E2 -8249.96} C_VEL
LIN {X 0,Y 454.863,Z 370.018,A -85,B 0,C 180,E1 -8250.56,E2 -8250.56} C_VEL
LIN {X 0,Y 455.172,Z 359.45,A -85,B 0,C 180,E1 -8251.089,E2 -8251.089} C_VEL
LIN {X 0,Y 455.283,Z 348.309,A -85,B 0,C 180,E1 -8251.458,E2 -8251.458} C_VEL
LIN {X 0,Y 455.498,Z 327.341,A -85,B 0,C 180,E1 -8251.839,E2 -8251.839} C_VEL
LIN {X 0,Y 455.882,Z 281.059,A -85,B 0,C 180,E1 -8252.609,E2 -8252.609} C_VEL
LIN {X 0,Y 453.644,Z 269.241,A -85,B 0,C 180,E1 -8252.899,E2 -8252.899} C_VEL
LIN {X 0,Y 453.528,Z 259.22,A -85,B 0,C 180,E1 -8255.023,E2 -8255.023} C_VEL
LIN {X 0,Y 453.468,Z 258.813,A -85,B 0,C 180,E1 -8255.142,E2 -8255.142} C_VEL
LIN {X 0,Y 453.468,Z 258.818,A -85,B 0,C 180,E1 -8258.416,E2 -8258.416} C_VEL
LIN {X 0,Y 453.511,Z 258.809,A -85,B 0,C 180,E1 -8261.009,E2 -8261.009} C_VEL
LIN {X 0,Y 453.557,Z 258.8,A -85,B 0,C 180,E1 -8263.88,E2 -8263.88} C_VEL
LIN {X 0,Y 453.552,Z 258.798,A -85,B 0,C 180,E1 -8267.472,E2 -8267.472} C_VEL
LIN {X 0,Y 453.583,Z 258.796,A -85,B 0,C 180,E1 -8271.087,E2 -8271.087} C_VEL
LIN {X 0,Y 453.67,Z 258.784,A -85,B 0,C 180,E1 -8273.775,E2 -8273.775} C_VEL
LIN {X 0,Y 453.757,Z 258.77,A -85,B 0,C 180,E1 -8277.338,E2 -8277.338} C_VEL
LIN {X 0,Y 453.814,Z 258.767,A -85,B 0,C 180,E1 -8280.001,E2 -8280.001} C_VEL
LIN {X 0,Y 453.757,Z 258.777,A -85,B 0,C 180,E1 -8282.664,E2 -8282.664} C_VEL
LIN {X 0,Y 453.669,Z 258.786,A -85,B 0,C 180,E1 -8286.226,E2 -8286.226} C_VEL
LIN {X 0,Y 453.584,Z 258.795,A -85,B 0,C 180,E1 -8288.914,E2 -8288.914} C_VEL
LIN {X 0,Y 453.555,Z 258.799,A -85,B 0,C 180,E1 -8292.53,E2 -8292.53} C_VEL
LIN {X 0,Y 453.537,Z 258.802,A -85,B 0,C 180,E1 -8296.197,E2 -8296.197} C_VEL
LIN {X 0,Y 453.513,Z 258.803,A -85,B 0,C 180,E1 -8299.042,E2 -8299.042} C_VEL
LIN {X 0,Y 453.469,Z 258.804,A -85,B 0,C 180,E1 -8301.837,E2 -8301.837} C_VEL
LIN {X 0,Y 453.508,Z 258.802,A -85,B 0,C 180,E1 -8304.735,E2 -8304.735} C_VEL
LIN {X 0,Y 453.532,Z 258.802,A -85,B 0,C 180,E1 -8307.962,E2 -8307.962} C_VEL
LIN {X 0,Y 453.477,Z 258.811,A -85,B 0,C 180,E1 -8310.76,E2 -8310.76} C_VEL
LIN {X 0,Y 453.472,Z 258.804,A -85,B 0,C 180,E1 -8313.914,E2 -8313.914} C_VEL
LIN {X 0,Y 453.466,Z 258.806,A -85,B 0,C 180,E1 -8317.189,E2 -8317.189} C_VEL
LIN {X 0,Y 453.526,Z 258.801,A -85,B 0,C 180,E1 -8319.446,E2 -8319.446} C_VEL
LIN {X 0,Y 453.457,Z 258.81,A -85,B 0,C 180,E1 -8322.996,E2 -8322.996} C_VEL
LIN {X 0,Y 453.462,Z 258.81,A -85,B 0,C 180,E1 -8325.78,E2 -8325.78} C_VEL
LIN {X 0,Y 453.476,Z 258.812,A -85,B 0,C 180,E1 -8328.21,E2 -8328.21} C_VEL
LIN {X 0,Y 453.512,Z 258.806,A -85,B 0,C 180,E1 -8330.791,E2 -8330.791} C_VEL
LIN {X 0,Y 453.454,Z 258.812,A -85,B 0,C 180,E1 -8333.918,E2 -8333.918} C_VEL
LIN {X 0,Y 453.481,Z 258.809,A -85,B 0,C 180,E1 -8337.152,E2 -8337.152} C_VEL
LIN {X 0,Y 453.473,Z 258.815,A -85,B 0,C 180,E1 -8340.269,E2 -8340.269} C_VEL
LIN {X 0,Y 453.5,Z 258.807,A -85,B 0,C 180,E1 -8343.294,E2 -8343.294} C_VEL
LIN {X 0,Y 453.564,Z 258.905,A -85,B 0,C 180,E1 -8345.349,E2 -8345.349} C_VEL
LIN {X 0,Y 454.782,Z 266.147,A -85,B 0,C 180,E1 -8346.793,E2 -8346.793} C_VEL
LIN {X 0,Y 454.395,Z 278.718,A -85,B 0,C 180,E1 -8349.162,E2 -8349.162} C_VEL
LIN {X 0,Y 453.848,Z 296.205,A -85,B 0,C 180,E1 -8352.425,E2 -8352.425} C_VEL
LIN {X 0,Y 453.396,Z 314.789,A -85,B 0,C 180,E1 -8355.87,E2 -8355.87} C_VEL
LIN {X 0,Y 453.341,Z 316.31,A -85,B 0,C 180,E1 -8356.14,E2 -8356.14} C_VEL
LIN {X 0,Y 455.644,Z 337.226,A -85,B 0,C 180,E1 -8356.568,E2 -8356.568} C_VEL
LIN {X 0,Y 455.15,Z 394.934,A -85,B 0,C 180,E1 -8357.544,E2 -8357.544} C_VEL
LIN {X 0,Y 454.821,Z 406.085,A -85,B 0,C 180,E1 -8357.875,E2 -8357.875} C_VEL
LIN {X 0,Y 454.398,Z 417.42,A -85,B 0,C 180,E1 -8358.401,E2 -8358.401} C_VEL
LIN {X 0,Y 454.09,Z 426.269,A -85,B 0,C 180,E1 -8358.958,E2 -8358.958} C_VEL
LIN {X 0,Y 453.75,Z 434.726,A -85,B 0,C 180,E1 -8359.627,E2 -8359.627} C_VEL
LIN {X 0,Y 453.448,Z 442.732,A -85,B 0,C 180,E1 -8360.409,E2 -8360.409} C_VEL
LIN {X 0,Y 453.118,Z 450.219,A -85,B 0,C 180,E1 -8361.302,E2 -8361.302} C_VEL
LIN {X 0,Y 452.88,Z 457.828,A -85,B 0,C 180,E1 -8362.421,E2 -8362.421} C_VEL
LIN {X 0,Y 452.652,Z 464.783,A -85,B 0,C 180,E1 -8363.761,E2 -8363.761} C_VEL
LIN {X 0,Y 452.582,Z 470.072,A -85,B 0,C 180,E1 -8365.101,E2 -8365.101} C_VEL
LIN {X 0,Y 452.557,Z 473.965,A -85,B 0,C 180,E1 -8366.439,E2 -8366.439} C_VEL
LIN {X 0,Y 452.55,Z 475.754,A -85,B 0,C 180,E1 -8367.33,E2 -8367.33} C_VEL
LIN {X 0,Y 452.511,Z 477.032,A -85,B 0,C 180,E1 -8368.22,E2 -8368.22} C_VEL
LIN {X 0,Y 452.494,Z 477.828,A -85,B 0,C 180,E1 -8369.11,E2 -8369.11} C_VEL
LIN {X 0,Y 452.476,Z 478.135,A -85,B 0,C 180,E1 -8370,E2 -8370} C_VEL
LIN {X 0,Y 452.494,Z 477.845,A -85,B 0,C 180,E1 -8370.89,E2 -8370.89} C_VEL
LIN {X 0,Y 452.511,Z 477.038,A -85,B 0,C 180,E1 -8371.78,E2 -8371.78} C_VEL
LIN {X 0,Y 452.551,Z 475.745,A -85,B 0,C 180,E1 -8372.67,E2 -8372.67} C_VEL
LIN {X 0,Y 452.526,Z 472.773,A -85,B 0,C 180,E1 -8374.008,E2 -8374.008} C_VEL
LIN {X 0,Y 452.619,Z 468.512,A -85,B 0,C 180,E1 -8375.346,E2 -8375.346} C_VEL
LIN {X 0,Y 452.729,Z 462.612,A -85,B 0,C 180,E1 -8376.686,E2 -8376.686} C_VEL
LIN {X 0,Y 452.881,Z 457.694,A -85,B 0,C 180,E1 -8377.58,E2 -8377.58} C_VEL
LIN {X 0,Y 453.064,Z 451.762,A -85,B 0,C 180,E1 -8378.474,E2 -8378.474} C_VEL
LIN {X 0,Y 453.345,Z 444.541,A -85,B 0,C 180,E1 -8379.368,E2 -8379.368} C_VEL
LIN {X 0,Y 453.677,Z 436.843,A -85,B 0,C 180,E1 -8380.149,E2 -8380.149} C_VEL
LIN {X 0,Y 453.999,Z 428.768,A -85,B 0,C 180,E1 -8380.818,E2 -8380.818} C_VEL
LIN {X 0,Y 454.262,Z 420.413,A -85,B 0,C 180,E1 -8381.377,E2 -8381.377} C_VEL
LIN {X 0,Y 454.55,Z 411.918,A -85,B 0,C 180,E1 -8381.822,E2 -8381.822} C_VEL
LIN {X 0,Y 454.868,Z 401.862,A -85,B 0,C 180,E1 -8382.209,E2 -8382.209} C_VEL
LIN {X 0,Y 455.139,Z 389.534,A -85,B 0,C 180,E1 -8382.502,E2 -8382.502} C_VEL
LIN {X 0,Y 455.371,Z 335.18,A -85,B 0,C 180,E1 -8383.395,E2 -8383.395} C_VEL
LIN {X 0,Y 453.337,Z 317.216,A -85,B 0,C 180,E1 -8383.778,E2 -8383.778} C_VEL
LIN {X 0,Y 453.827,Z 302.256,A -85,B 0,C 180,E1 -8386.648,E2 -8386.648} C_VEL
LIN {X 0,Y 454.507,Z 284.29,A -85,B 0,C 180,E1 -8390.124,E2 -8390.124} C_VEL
LIN {X 0,Y 455.172,Z 268.684,A -85,B 0,C 180,E1 -8393.186,E2 -8393.186} C_VEL
LIN {X 0,Y 453.549,Z 258.804,A -85,B 0,C 180,E1 -8395.283,E2 -8395.283} C_VEL
LIN {X 0,Y 453.508,Z 258.804,A -85,B 0,C 180,E1 -8398.712,E2 -8398.712} C_VEL
LIN {X 0,Y 453.464,Z 258.812,A -85,B 0,C 180,E1 -8401.799,E2 -8401.799} C_VEL
LIN {X 0,Y 453.48,Z 258.807,A -85,B 0,C 180,E1 -8404.989,E2 -8404.989} C_VEL
LIN {X 0,Y 453.464,Z 258.808,A -85,B 0,C 180,E1 -8408.311,E2 -8408.311} C_VEL
LIN {X 0,Y 453.493,Z 258.804,A -85,B 0,C 180,E1 -8410.608,E2 -8410.608} C_VEL
LIN {X 0,Y 453.455,Z 258.813,A -85,B 0,C 180,E1 -8413.244,E2 -8413.244} C_VEL
LIN {X 0,Y 453.463,Z 258.812,A -85,B 0,C 180,E1 -8415.778,E2 -8415.778} C_VEL
LIN {X 0,Y 453.477,Z 258.807,A -85,B 0,C 180,E1 -8418.209,E2 -8418.209} C_VEL
LIN {X 0,Y 453.485,Z 258.805,A -85,B 0,C 180,E1 -8420.794,E2 -8420.794} C_VEL
LIN {X 0,Y 453.454,Z 258.812,A -85,B 0,C 180,E1 -8423.917,E2 -8423.917} C_VEL
LIN {X 0,Y 453.48,Z 258.809,A -85,B 0,C 180,E1 -8427.15,E2 -8427.15} C_VEL
LIN {X 0,Y 453.471,Z 258.807,A -85,B 0,C 180,E1 -8430.268,E2 -8430.268} C_VEL
LIN {X 0,Y 453.511,Z 258.806,A -85,B 0,C 180,E1 -8433.294,E2 -8433.294} C_VEL
LIN {X 0,Y 453.5,Z 258.804,A -85,B 0,C 180,E1 -8436.238,E2 -8436.238} C_VEL
LIN {X 0,Y 453.478,Z 258.808,A -85,B 0,C 180,E1 -8439.117,E2 -8439.117} C_VEL
LIN {X 0,Y 453.507,Z 258.805,A -85,B 0,C 180,E1 -8441.944,E2 -8441.944} C_VEL
LIN {X 0,Y 453.535,Z 258.799,A -85,B 0,C 180,E1 -8444.726,E2 -8444.726} C_VEL
LIN {X 0,Y 453.554,Z 258.797,A -85,B 0,C 180,E1 -8448.378,E2 -8448.378} C_VEL
LIN {X 0,Y 453.647,Z 258.788,A -85,B 0,C 180,E1 -8451.984,E2 -8451.984} C_VEL
LIN {X 0,Y 453.665,Z 258.783,A -85,B 0,C 180,E1 -8454.666,E2 -8454.666} C_VEL
LIN {X 0,Y 453.759,Z 258.776,A -85,B 0,C 180,E1 -8457.336,E2 -8457.336} C_VEL
LIN {X 0,Y 453.817,Z 258.766,A -85,B 0,C 180,E1 -8459.999,E2 -8459.999} C_VEL
LIN {X 0,Y 453.759,Z 258.771,A -85,B 0,C 180,E1 -8462.662,E2 -8462.662} C_VEL
LIN {X 0,Y 453.67,Z 258.783,A -85,B 0,C 180,E1 -8466.225,E2 -8466.225} C_VEL
LIN {X 0,Y 453.585,Z 258.794,A -85,B 0,C 180,E1 -8468.913,E2 -8468.913} C_VEL
LIN {X 0,Y 453.594,Z 258.792,A -85,B 0,C 180,E1 -8472.55,E2 -8472.55} C_VEL
LIN {X 0,Y 453.537,Z 258.8,A -85,B 0,C 180,E1 -8476.195,E2 -8476.195} C_VEL
LIN {X 0,Y 453.512,Z 258.804,A -85,B 0,C 180,E1 -8479.04,E2 -8479.04} C_VEL
LIN {X 0,Y 453.468,Z 258.812,A -85,B 0,C 180,E1 -8481.836,E2 -8481.836} C_VEL
LIN {X 0,Y 453.506,Z 258.803,A -85,B 0,C 180,E1 -8484.734,E2 -8484.734} C_VEL
LIN {X 0,Y 453.529,Z 258.803,A -85,B 0,C 180,E1 -8487.96,E2 -8487.96} C_VEL
LIN {X 0,Y 453.458,Z 258.815,A -85,B 0,C 180,E1 -8491.525,E2 -8491.525} C_VEL
LIN {X 0,Y 453.48,Z 258.807,A -85,B 0,C 180,E1 -8494.777,E2 -8494.777} C_VEL
LIN {X 0,Y 453.475,Z 258.807,A -85,B 0,C 180,E1 -8498.309,E2 -8498.309} C_VEL
LIN {X 0,Y 453.507,Z 258.803,A -85,B 0,C 180,E1 -8500.606,E2 -8500.606} C_VEL
LIN {X 0,Y 453.464,Z 258.809,A -85,B 0,C 180,E1 -8504.22,E2 -8504.22} C_VEL
LIN {X 0,Y 453.482,Z 258.807,A -85,B 0,C 180,E1 -8507.008,E2 -8507.008} C_VEL
LIN {X 0,Y 453.519,Z 258.801,A -85,B 0,C 180,E1 -8510.554,E2 -8510.554} C_VEL
LIN {X 0,Y 453.447,Z 258.814,A -85,B 0,C 180,E1 -8513.917,E2 -8513.917} C_VEL
LIN {X 0,Y 453.474,Z 258.809,A -85,B 0,C 180,E1 -8517.151,E2 -8517.151} C_VEL
LIN {X 0,Y 453.465,Z 258.809,A -85,B 0,C 180,E1 -8520.268,E2 -8520.268} C_VEL
LIN {X 0,Y 453.497,Z 258.807,A -85,B 0,C 180,E1 -8523.294,E2 -8523.294} C_VEL
LIN {X 0,Y 453.496,Z 258.805,A -85,B 0,C 180,E1 -8526.239,E2 -8526.239} C_VEL
LIN {X 0,Y 453.484,Z 258.808,A -85,B 0,C 180,E1 -8529.118,E2 -8529.118} C_VEL
LIN {X 0,Y 453.503,Z 258.807,A -85,B 0,C 180,E1 -8531.944,E2 -8531.944} C_VEL
LIN {X 0,Y 453.531,Z 258.8,A -85,B 0,C 180,E1 -8534.726,E2 -8534.726} C_VEL
LIN {X 0,Y 453.552,Z 258.798,A -85,B 0,C 180,E1 -8538.379,E2 -8538.379} C_VEL
LIN {X 0,Y 453.643,Z 258.789,A -85,B 0,C 180,E1 -8541.985,E2 -8541.985} C_VEL
LIN {X 0,Y 453.619,Z 258.79,A -85,B 0,C 180,E1 -8543.097,E2 -8543.097} C_VEL
LIN {X 0,Y 452.935,Z 258.879,A -85,B 0,C 180,E1 -8543.838,E2 -8543.838} C_VEL
LIN {X 0,Y 449.991,Z 259.242,A -85,B 0,C 180,E1 -8545.039,E2 -8545.039} C_VEL
LIN {X 0,Y 447.568,Z 259.546,A -85,B 0,C 180,E1 -8546.009,E2 -8546.009} C_VEL
LIN {X 0,Y 446.625,Z 259.661,A -85,B 0,C 180,E1 -8546.759,E2 -8546.759} C_VEL
LIN {X 0,Y 446.602,Z 259.664,A -85,B 0,C 180,E1 -8547.013,E2 -8547.013} C_VEL
LIN {X 0,Y 446.783,Z 259.644,A -85,B 0,C 180,E1 -8550,E2 -8550} C_VEL
LIN {X 0,Y 446.681,Z 259.654,A -85,B 0,C 180,E1 -8552.705,E2 -8552.705} C_VEL
LIN {X 0,Y 446.626,Z 259.661,A -85,B 0,C 180,E1 -8556.324,E2 -8556.324} C_VEL
LIN {X 0,Y 446.528,Z 259.674,A -85,B 0,C 180,E1 -8559.055,E2 -8559.055} C_VEL
LIN {X 0,Y 446.524,Z 259.674,A -85,B 0,C 180,E1 -8562.729,E2 -8562.729} C_VEL
LIN {X 0,Y 446.479,Z 259.679,A -85,B 0,C 180,E1 -8566.459,E2 -8566.459} C_VEL
LIN {X 0,Y 446.458,Z 259.684,A -85,B 0,C 180,E1 -8569.303,E2 -8569.303} C_VEL
LIN {X 0,Y 446.406,Z 259.689,A -85,B 0,C 180,E1 -8572.199,E2 -8572.199} C_VEL
LIN {X 0,Y 446.428,Z 259.687,A -85,B 0,C 180,E1 -8575.153,E2 -8575.153} C_VEL
LIN {X 0,Y 446.474,Z 259.681,A -85,B 0,C 180,E1 -8578.179,E2 -8578.179} C_VEL
LIN {X 0,Y 446.414,Z 259.694,A -85,B 0,C 180,E1 -8581.776,E2 -8581.776} C_VEL
LIN {X 0,Y 446.48,Z 259.871,A -85,B 0,C 180,E1 -8582.623,E2 -8582.623} C_VEL
LIN {X 0,Y 446.567,Z 266.197,A -85,B 0,C 180,E1 -8584.236,E2 -8584.236} C_VEL
LIN {X 0,Y 446.496,Z 269.731,A -85,B 0,C 180,E1 -8585.119,E2 -8585.119} C_VEL
LIN {X 0,Y 448.826,Z 283.421,A -85,B 0,C 180,E1 -8585.43,E2 -8585.43} C_VEL
LIN {X 0,Y 448.242,Z 345.737,A -85,B 0,C 180,E1 -8586.492,E2 -8586.492} C_VEL
LIN {X 0,Y 448.027,Z 355.684,A -85,B 0,C 180,E1 -8586.783,E2 -8586.783} C_VEL
LIN {X 0,Y 447.874,Z 367.665,A -85,B 0,C 180,E1 -8587.321,E2 -8587.321} C_VEL
LIN {X 0,Y 447.528,Z 376.61,A -85,B 0,C 180,E1 -8587.881,E2 -8587.881} C_VEL
LIN {X 0,Y 447.258,Z 385.123,A -85,B 0,C 180,E1 -8588.558,E2 -8588.558} C_VEL
LIN {X 0,Y 446.96,Z 392.489,A -85,B 0,C 180,E1 -8589.275,E2 -8589.275} C_VEL
LIN {X 0,Y 446.585,Z 400.115,A -85,B 0,C 180,E1 -8590.181,E2 -8590.181} C_VEL
LIN {X 0,Y 446.351,Z 406.603,A -85,B 0,C 180,E1 -8591.126,E2 -8591.126} C_VEL
LIN {X 0,Y 446.057,Z 412.767,A -85,B 0,C 180,E1 -8592.226,E2 -8592.226} C_VEL
LIN {X 0,Y 445.839,Z 418.493,A -85,B 0,C 180,E1 -8593.523,E2 -8593.523} C_VEL
LIN {X 0,Y 445.669,Z 422.633,A -85,B 0,C 180,E1 -8594.797,E2 -8594.797} C_VEL
LIN {X 0,Y 445.475,Z 426.436,A -85,B 0,C 180,E1 -8596.527,E2 -8596.527} C_VEL
LIN {X 0,Y 445.389,Z 428.087,A -85,B 0,C 180,E1 -8597.869,E2 -8597.869} C_VEL
LIN {X 0,Y 445.387,Z 428.555,A -85,B 0,C 180,E1 -8599.235,E2 -8599.235} C_VEL
LIN {X 0,Y 445.42,Z 427.576,A -85,B 0,C 180,E1 -8600.868,E2 -8600.868} C_VEL
LIN {X 0,Y 445.622,Z 424.761,A -85,B 0,C 180,E1 -8602.626,E2 -8602.626} C_VEL
LIN {X 0,Y 445.809,Z 421.246,A -85,B 0,C 180,E1 -8603.922,E2 -8603.922} C_VEL
LIN {X 0,Y 446.026,Z 417.301,A -85,B 0,C 180,E1 -8605.019,E2 -8605.019} C_VEL
LIN {X 0,Y 446.222,Z 412.871,A -85,B 0,C 180,E1 -8606.006,E2 -8606.006} C_VEL
LIN {X 0,Y 446.456,Z 406.735,A -85,B 0,C 180,E1 -8607.107,E2 -8607.107} C_VEL
LIN {X 0,Y 446.8,Z 399.553,A -85,B 0,C 180,E1 -8608.144,E2 -8608.144} C_VEL
LIN {X 0,Y 447.257,Z 390.816,A -85,B 0,C 180,E1 -8609.155,E2 -8609.155} C_VEL
LIN {X 0,Y 447.639,Z 381.708,A -85,B 0,C 180,E1 -8609.972,E2 -8609.972} C_VEL
LIN {X 0,Y 447.852,Z 373.396,A -85,B 0,C 180,E1 -8610.57,E2 -8610.57} C_VEL
LIN {X 0,Y 448.096,Z 364.87,A -85,B 0,C 180,E1 -8611.052,E2 -8611.052} C_VEL
LIN {X 0,Y 448.322,Z 355.098,A -85,B 0,C 180,E1 -8611.463,E2 -8611.463} C_VEL
LIN {X 0,Y 448.439,Z 345.809,A -85,B 0,C 180,E1 -8611.728,E2 -8611.728} C_VEL
LIN {X 0,Y 449.081,Z 282.146,A -85,B 0,C 180,E1 -8612.822,E2 -8612.822} C_VEL
LIN {X 0,Y 446.669,Z 269.627,A -85,B 0,C 180,E1 -8613.135,E2 -8613.135} C_VEL
LIN {X 0,Y 446.563,Z 260.462,A -85,B 0,C 180,E1 -8615.104,E2 -8615.104} C_VEL
LIN {X 0,Y 446.443,Z 259.688,A -85,B 0,C 180,E1 -8615.345,E2 -8615.345} C_VEL
LIN {X 0,Y 446.441,Z 259.693,A -85,B 0,C 180,E1 -8618.774,E2 -8618.774} C_VEL
LIN {X 0,Y 446.446,Z 259.687,A -85,B 0,C 180,E1 -8621.65,E2 -8621.65} C_VEL
LIN {X 0,Y 446.496,Z 259.683,A -85,B 0,C 180,E1 -8624.48,E2 -8624.48} C_VEL
LIN {X 0,Y 446.508,Z 259.679,A -85,B 0,C 180,E1 -8628.194,E2 -8628.194} C_VEL
LIN {X 0,Y 446.59,Z 259.667,A -85,B 0,C 180,E1 -8631.858,E2 -8631.858} C_VEL
LIN {X 0,Y 446.639,Z 259.663,A -85,B 0,C 180,E1 -8634.583,E2 -8634.583} C_VEL
LIN {X 0,Y 446.701,Z 259.649,A -85,B 0,C 180,E1 -8637.295,E2 -8637.295} C_VEL
LIN {X 0,Y 446.784,Z 259.643,A -85,B 0,C 180,E1 -8640.001,E2 -8640.001} C_VEL
LIN {X 0,Y 446.701,Z 259.656,A -85,B 0,C 180,E1 -8642.706,E2 -8642.706} C_VEL
LIN {X 0,Y 446.638,Z 259.664,A -85,B 0,C 180,E1 -8646.325,E2 -8646.325} C_VEL
LIN {X 0,Y 446.53,Z 259.673,A -85,B 0,C 180,E1 -8649.056,E2 -8649.056} C_VEL
LIN {X 0,Y 446.513,Z 259.676,A -85,B 0,C 180,E1 -8652.731,E2 -8652.731} C_VEL
LIN {X 0,Y 446.488,Z 259.68,A -85,B 0,C 180,E1 -8656.229,E2 -8656.229} C_VEL
LIN {X 0,Y 446.462,Z 259.68,A -85,B 0,C 180,E1 -8659.304,E2 -8659.304} C_VEL
LIN {X 0,Y 446.411,Z 259.687,A -85,B 0,C 180,E1 -8662.201,E2 -8662.201} C_VEL
LIN {X 0,Y 446.451,Z 259.678,A -85,B 0,C 180,E1 -8665.153,E2 -8665.153} C_VEL
LIN {X 0,Y 446.478,Z 259.682,A -85,B 0,C 180,E1 -8668.18,E2 -8668.18} C_VEL
LIN {X 0,Y 446.413,Z 259.687,A -85,B 0,C 180,E1 -8671.301,E2 -8671.301} C_VEL
LIN {X 0,Y 446.425,Z 259.689,A -85,B 0,C 180,E1 -8674.524,E2 -8674.524} C_VEL
LIN {X 0,Y 446.432,Z 259.684,A -85,B 0,C 180,E1 -8678.084,E2 -8678.084} C_VEL
LIN {X 0,Y 446.439,Z 259.686,A -85,B 0,C 180,E1 -8680.921,E2 -8680.921} C_VEL
LIN {X 0,Y 446.396,Z 259.688,A -85,B 0,C 180,E1 -8683.847,E2 -8683.847} C_VEL
LIN {X 0,Y 446.396,Z 259.693,A -85,B 0,C 180,E1 -8686.404,E2 -8686.404} C_VEL
LIN {X 0,Y 446.424,Z 259.687,A -85,B 0,C 180,E1 -8689.083,E2 -8689.083} C_VEL
LIN {X 0,Y 446.427,Z 259.687,A -85,B 0,C 180,E1 -8691.919,E2 -8691.919} C_VEL
LIN {X 0,Y 446.428,Z 259.686,A -85,B 0,C 180,E1 -8695.478,E2 -8695.478} C_VEL
LIN {X 0,Y 446.415,Z 259.693,A -85,B 0,C 180,E1 -8698.701,E2 -8698.701} C_VEL
LIN {X 0,Y 446.484,Z 259.683,A -85,B 0,C 180,E1 -8701.822,E2 -8701.822} C_VEL
LIN {X 0,Y 446.503,Z 259.684,A -85,B 0,C 180,E1 -8705.162,E2 -8705.162} C_VEL
LIN {X 0,Y 447.865,Z 268.282,A -85,B 0,C 180,E1 -8706.903,E2 -8706.903} C_VEL
LIN {X 0,Y 447.316,Z 283.36,A -85,B 0,C 180,E1 -8709.779,E2 -8709.779} C_VEL
LIN {X 0,Y 446.669,Z 302.061,A -85,B 0,C 180,E1 -8713.313,E2 -8713.313} C_VEL
LIN {X 0,Y 446.347,Z 315.69,A -85,B 0,C 180,E1 -8715.875,E2 -8715.875} C_VEL
LIN {X 0,Y 448.751,Z 337.956,A -85,B 0,C 180,E1 -8716.362,E2 -8716.362} C_VEL
LIN {X 0,Y 448.211,Z 393.788,A -85,B 0,C 180,E1 -8717.32,E2 -8717.32} C_VEL
LIN {X 0,Y 447.991,Z 403.538,A -85,B 0,C 180,E1 -8717.601,E2 -8717.601} C_VEL
LIN {X 0,Y 447.616,Z 414.084,A -85,B 0,C 180,E1 -8718.051,E2 -8718.051} C_VEL
LIN {X 0,Y 447.191,Z 424.493,A -85,B 0,C 180,E1 -8718.671,E2 -8718.671} C_VEL
LIN {X 0,Y 446.747,Z 434.423,A -85,B 0,C 180,E1 -8719.463,E2 -8719.463} C_VEL
LIN {X 0,Y 446.412,Z 442.402,A -85,B 0,C 180,E1 -8720.257,E2 -8720.257} C_VEL
LIN {X 0,Y 446.087,Z 449.872,A -85,B 0,C 180,E1 -8721.164,E2 -8721.164} C_VEL
LIN {X 0,Y 445.814,Z 457.464,A -85,B 0,C 180,E1 -8722.3,E2 -8722.3} C_VEL
LIN {X 0,Y 445.569,Z 464.01,A -85,B 0,C 180,E1 -8723.569,E2 -8723.569} C_VEL
LIN {X 0,Y 445.512,Z 469.695,A -85,B 0,C 180,E1 -8725.023,E2 -8725.023} C_VEL
LIN {X 0,Y 445.455,Z 473.585,A -85,B 0,C 180,E1 -8726.382,E2 -8726.382} C_VEL
LIN {X 0,Y 445.475,Z 475.373,A -85,B 0,C 180,E1 -8727.287,E2 -8727.287} C_VEL
LIN {X 0,Y 445.426,Z 476.647,A -85,B 0,C 180,E1 -8728.192,E2 -8728.192} C_VEL
LIN {X 0,Y 445.431,Z 477.438,A -85,B 0,C 180,E1 -8729.096,E2 -8729.096} C_VEL
LIN {X 0,Y 445.411,Z 477.742,A -85,B 0,C 180,E1 -8730,E2 -8730} C_VEL
LIN {X 0,Y 445.43,Z 477.452,A -85,B 0,C 180,E1 -8730.904,E2 -8730.904} C_VEL
LIN {X 0,Y 445.426,Z 476.636,A -85,B 0,C 180,E1 -8731.809,E2 -8731.809} C_VEL
LIN {X 0,Y 445.476,Z 475.335,A -85,B 0,C 180,E1 -8732.713,E2 -8732.713} C_VEL
LIN {X 0,Y 445.43,Z 472.351,A -85,B 0,C 180,E1 -8734.072,E2 -8734.072} C_VEL
LIN {X 0,Y 445.532,Z 468.078,A -85,B 0,C 180,E1 -8735.431,E2 -8735.431} C_VEL
LIN {X 0,Y 445.656,Z 462.151,A -85,B 0,C 180,E1 -8736.792,E2 -8736.792} C_VEL
LIN {X 0,Y 445.812,Z 457.215,A -85,B 0,C 180,E1 -8737.701,E2 -8737.701} C_VEL
LIN {X 0,Y 446.021,Z 451.263,A -85,B 0,C 180,E1 -8738.609,E2 -8738.609} C_VEL
LIN {X 0,Y 446.345,Z 444.019,A -85,B 0,C 180,E1 -8739.516,E2 -8739.516} C_VEL
LIN {X 0,Y 446.657,Z 436.289,A -85,B 0,C 180,E1 -8740.31,E2 -8740.31} C_VEL
LIN {X 0,Y 446.996,Z 428.176,A -85,B 0,C 180,E1 -8740.99,E2 -8740.99} C_VEL
LIN {X 0,Y 447.29,Z 419.771,A -85,B 0,C 180,E1 -8741.556,E2 -8741.556} C_VEL
LIN {X 0,Y 447.568,Z 411.202,A -85,B 0,C 180,E1 -8742.009,E2 -8742.009} C_VEL
LIN {X 0,Y 447.934,Z 401.033,A -85,B 0,C 180,E1 -8742.401,E2 -8742.401} C_VEL
LIN {X 0,Y 448.179,Z 387.317,A -85,B 0,C 180,E1 -8742.714,E2 -8742.714} C_VEL
LIN {X 0,Y 448.414,Z 335.48,A -85,B 0,C 180,E1 -8743.583,E2 -8743.583} C_VEL
LIN {X 0,Y 446.313,Z 316.878,A -85,B 0,C 180,E1 -8743.982,E2 -8743.982} C_VEL
LIN {X 0,Y 446.916,Z 299.426,A -85,B 0,C 180,E1 -8747.385,E2 -8747.385} C_VEL
LIN {X 0,Y 447.64,Z 281.475,A -85,B 0,C 180,E1 -8750.927,E2 -8750.927} C_VEL
LIN {X 0,Y 448.163,Z 269.455,A -85,B 0,C 180,E1 -8753.326,E2 -8753.326} C_VEL
LIN {X 0,Y 446.486,Z 259.685,A -85,B 0,C 180,E1 -8755.431,E2 -8755.431} C_VEL
LIN {X 0,Y 446.486,Z 259.679,A -85,B 0,C 180,E1 -8758.178,E2 -8758.178} C_VEL
LIN {X 0,Y 446.419,Z 259.69,A -85,B 0,C 180,E1 -8761.774,E2 -8761.774} C_VEL
LIN {X 0,Y 446.429,Z 259.684,A -85,B 0,C 180,E1 -8764.522,E2 -8764.522} C_VEL
LIN {X 0,Y 446.415,Z 259.687,A -85,B 0,C 180,E1 -8768.079,E2 -8768.079} C_VEL
LIN {X 0,Y 446.426,Z 259.685,A -85,B 0,C 180,E1 -8770.917,E2 -8770.917} C_VEL
LIN {X 0,Y 446.4,Z 259.691,A -85,B 0,C 180,E1 -8773.845,E2 -8773.845} C_VEL
LIN {X 0,Y 446.396,Z 259.688,A -85,B 0,C 180,E1 -8776.403,E2 -8776.403} C_VEL
LIN {X 0,Y 446.425,Z 259.687,A -85,B 0,C 180,E1 -8779.082,E2 -8779.082} C_VEL
LIN {X 0,Y 446.406,Z 259.688,A -85,B 0,C 180,E1 -8782.12,E2 -8782.12} C_VEL
LIN {X 0,Y 446.428,Z 259.691,A -85,B 0,C 180,E1 -8785.476,E2 -8785.476} C_VEL
LIN {X 0,Y 446.412,Z 259.686,A -85,B 0,C 180,E1 -8788.699,E2 -8788.699} C_VEL
LIN {X 0,Y 446.481,Z 259.682,A -85,B 0,C 180,E1 -8791.821,E2 -8791.821} C_VEL
LIN {X 0,Y 446.455,Z 259.682,A -85,B 0,C 180,E1 -8794.847,E2 -8794.847} C_VEL
LIN {X 0,Y 446.444,Z 259.683,A -85,B 0,C 180,E1 -8798.244,E2 -8798.244} C_VEL
LIN {X 0,Y 446.453,Z 259.688,A -85,B 0,C 180,E1 -8801.648,E2 -8801.648} C_VEL
LIN {X 0,Y 446.503,Z 259.675,A -85,B 0,C 180,E1 -8804.479,E2 -8804.479} C_VEL
LIN {X 0,Y 446.512,Z 259.675,A -85,B 0,C 180,E1 -8808.192,E2 -8808.192} C_VEL
LIN {X 0,Y 446.595,Z 259.668,A -85,B 0,C 180,E1 -8811.857,E2 -8811.857} C_VEL
LIN {X 0,Y 446.64,Z 259.658,A -85,B 0,C 180,E1 -8814.582,E2 -8814.582} C_VEL
LIN {X 0,Y 446.703,Z 259.654,A -85,B 0,C 180,E1 -8817.294,E2 -8817.294} C_VEL
LIN {X 0,Y 446.787,Z 259.642,A -85,B 0,C 180,E1 -8819.999,E2 -8819.999} C_VEL
LIN {X 0,Y 446.703,Z 259.65,A -85,B 0,C 180,E1 -8822.705,E2 -8822.705} C_VEL
LIN {X 0,Y 446.639,Z 259.659,A -85,B 0,C 180,E1 -8826.323,E2 -8826.323} C_VEL
LIN {X 0,Y 446.531,Z 259.673,A -85,B 0,C 180,E1 -8829.055,E2 -8829.055} C_VEL
LIN {X 0,Y 446.526,Z 259.673,A -85,B 0,C 180,E1 -8832.729,E2 -8832.729} C_VEL
LIN {X 0,Y 446.482,Z 259.678,A -85,B 0,C 180,E1 -8836.458,E2 -8836.458} C_VEL
LIN {X 0,Y 446.461,Z 259.684,A -85,B 0,C 180,E1 -8839.303,E2 -8839.303} C_VEL
LIN {X 0,Y 446.409,Z 259.688,A -85,B 0,C 180,E1 -8842.199,E2 -8842.199} C_VEL
LIN {X 0,Y 446.45,Z 259.684,A -85,B 0,C 180,E1 -8845.152,E2 -8845.152} C_VEL
LIN {X 0,Y 446.476,Z 259.68,A -85,B 0,C 180,E1 -8848.178,E2 -8848.178} C_VEL
LIN {X 0,Y 446.411,Z 259.692,A -85,B 0,C 180,E1 -8851.775,E2 -8851.775} C_VEL
LIN {X 0,Y 446.421,Z 259.686,A -85,B 0,C 180,E1 -8854.522,E2 -8854.522} C_VEL
LIN {X 0,Y 446.429,Z 259.687,A -85,B 0,C 180,E1 -8858.083,E2 -8858.083} C_VEL
LIN {X 0,Y 446.435,Z 259.685,A -85,B 0,C 180,E1 -8860.92,E2 -8860.92} C_VEL
LIN {X 0,Y 446.413,Z 259.691,A -85,B 0,C 180,E1 -8863.843,E2 -8863.843} C_VEL
LIN {X 0,Y 446.437,Z 259.684,A -85,B 0,C 180,E1 -8866.397,E2 -8866.397} C_VEL
LIN {X 0,Y 446.458,Z 259.686,A -85,B 0,C 180,E1 -8869.804,E2 -8869.804} C_VEL
LIN {X 0,Y 446.422,Z 259.687,A -85,B 0,C 180,E1 -8872.123,E2 -8872.123} C_VEL
LIN {X 0,Y 446.421,Z 259.691,A -85,B 0,C 180,E1 -8875.477,E2 -8875.477} C_VEL
LIN {X 0,Y 446.407,Z 259.688,A -85,B 0,C 180,E1 -8878.699,E2 -8878.699} C_VEL
LIN {X 0,Y 446.475,Z 259.684,A -85,B 0,C 180,E1 -8881.821,E2 -8881.821} C_VEL
LIN {X 0,Y 446.449,Z 259.683,A -85,B 0,C 180,E1 -8884.848,E2 -8884.848} C_VEL
LIN {X 0,Y 446.441,Z 259.684,A -85,B 0,C 180,E1 -8888.244,E2 -8888.244} C_VEL
LIN {X 0,Y 446.449,Z 259.689,A -85,B 0,C 180,E1 -8891.649,E2 -8891.649} C_VEL
LIN {X 0,Y 446.499,Z 259.676,A -85,B 0,C 180,E1 -8894.48,E2 -8894.48} C_VEL
LIN {X 0,Y 446.51,Z 259.676,A -85,B 0,C 180,E1 -8898.193,E2 -8898.193} C_VEL
LIN {X 0,Y 446.591,Z 259.669,A -85,B 0,C 180,E1 -8901.858,E2 -8901.858} C_VEL
LIN {X 0,Y 446.631,Z 259.66,A -85,B 0,C 180,E1 -8904.582,E2 -8904.582} C_VEL
LIN {X 0,Y 446.602,Z 259.664,A -85,B 0,C 180,E1 -8907.013,E2 -8907.013} C_VEL
LIN {X 0,Y 446.078,Z 259.734,A -85,B 0,C 180,E1 -8907.766,E2 -8907.766} C_VEL
LIN {X 0,Y 443.266,Z 260.084,A -85,B 0,C 180,E1 -8908.989,E2 -8908.989} C_VEL
LIN {X 0,Y 440.79,Z 260.391,A -85,B 0,C 180,E1 -8909.976,E2 -8909.976} C_VEL
LIN {X 0,Y 439.706,Z 260.524,A -85,B 0,C 180,E1 -8910.74,E2 -8910.74} C_VEL
LIN {X 0,Y 439.612,Z 260.535,A -85,B 0,C 180,E1 -8910.998,E2 -8910.998} C_VEL
LIN {X 0,Y 439.631,Z 260.532,A -85,B 0,C 180,E1 -8912.749,E2 -8912.749} C_VEL
LIN {X 0,Y 439.601,Z 260.536,A -85,B 0,C 180,E1 -8916.425,E2 -8916.425} C_VEL
LIN {X 0,Y 439.49,Z 260.551,A -85,B 0,C 180,E1 -8919.201,E2 -8919.201} C_VEL
LIN {X 0,Y 439.494,Z 260.549,A -85,B 0,C 180,E1 -8922.726,E2 -8922.726} C_VEL
LIN {X 0,Y 439.437,Z 260.557,A -85,B 0,C 180,E1 -8926.348,E2 -8926.348} C_VEL
LIN {X 0,Y 439.392,Z 260.567,A -85,B 0,C 180,E1 -8929.626,E2 -8929.626} C_VEL
LIN {X 0,Y 439.352,Z 260.567,A -85,B 0,C 180,E1 -8932.575,E2 -8932.575} C_VEL
LIN {X 0,Y 439.376,Z 260.569,A -85,B 0,C 180,E1 -8935.586,E2 -8935.586} C_VEL
LIN {X 0,Y 439.405,Z 260.56,A -85,B 0,C 180,E1 -8938.673,E2 -8938.673} C_VEL
LIN {X 0,Y 439.442,Z 260.634,A -85,B 0,C 180,E1 -8942.503,E2 -8942.503} C_VEL
LIN {X 0,Y 439.537,Z 267.662,A -85,B 0,C 180,E1 -8944.306,E2 -8944.306} C_VEL
LIN {X 0,Y 439.49,Z 270.029,A -85,B 0,C 180,E1 -8944.902,E2 -8944.902} C_VEL
LIN {X 0,Y 441.902,Z 283.187,A -85,B 0,C 180,E1 -8945.222,E2 -8945.222} C_VEL
LIN {X 0,Y 441.303,Z 346.106,A -85,B 0,C 180,E1 -8946.314,E2 -8946.314} C_VEL
LIN {X 0,Y 441.073,Z 355.851,A -85,B 0,C 180,E1 -8946.602,E2 -8946.602} C_VEL
LIN {X 0,Y 440.912,Z 366.257,A -85,B 0,C 180,E1 -8947.062,E2 -8947.062} C_VEL
LIN {X 0,Y 440.541,Z 377.274,A -85,B 0,C 180,E1 -8947.748,E2 -8947.748} C_VEL
LIN {X 0,Y 440.23,Z 386.487,A -85,B 0,C 180,E1 -8948.506,E2 -8948.506} C_VEL
LIN {X 0,Y 439.908,Z 394.047,A -85,B 0,C 180,E1 -8949.274,E2 -8949.274} C_VEL
LIN {X 0,Y 439.562,Z 400.878,A -85,B 0,C 180,E1 -8950.114,E2 -8950.114} C_VEL
LIN {X 0,Y 439.244,Z 408.325,A -85,B 0,C 180,E1 -8951.237,E2 -8951.237} C_VEL
LIN {X 0,Y 438.923,Z 415.181,A -85,B 0,C 180,E1 -8952.564,E2 -8952.564} C_VEL
LIN {X 0,Y 438.755,Z 419.153,A -85,B 0,C 180,E1 -8953.532,E2 -8953.532} C_VEL
LIN {X 0,Y 438.577,Z 423.238,A -85,B 0,C 180,E1 -8954.835,E2 -8954.835} C_VEL
LIN {X 0,Y 438.412,Z 426.218,A -85,B 0,C 180,E1 -8956.167,E2 -8956.167} C_VEL
LIN {X 0,Y 438.308,Z 428.272,A -85,B 0,C 180,E1 -8957.668,E2 -8957.668} C_VEL
LIN {X 0,Y 438.288,Z 428.927,A -85,B 0,C 180,E1 -8958.906,E2 -8958.906} C_VEL
LIN {X 0,Y 438.311,Z 428.567,A -85,B 0,C 180,E1 -8960.32,E2 -8960.32} C_VEL
LIN {X 0,Y 438.428,Z 426.874,A -85,B 0,C 180,E1 -8961.762,E2 -8961.762} C_VEL
LIN {X 0,Y 438.522,Z 425.619,A -85,B 0,C 180,E1 -8962.484,E2 -8962.484} C_VEL
LIN {X 0,Y 438.705,Z 422.79,A -85,B 0,C 180,E1 -8963.65,E2 -8963.65} C_VEL
LIN {X 0,Y 438.969,Z 417.88,A -85,B 0,C 180,E1 -8965.086,E2 -8965.086} C_VEL
LIN {X 0,Y 439.243,Z 412.398,A -85,B 0,C 180,E1 -8966.304,E2 -8966.304} C_VEL
LIN {X 0,Y 439.453,Z 406.892,A -85,B 0,C 180,E1 -8967.289,E2 -8967.289} C_VEL
LIN {X 0,Y 439.763,Z 400.913,A -85,B 0,C 180,E1 -8968.172,E2 -8968.172} C_VEL
LIN {X 0,Y 440.151,Z 394.095,A -85,B 0,C 180,E1 -8969.008,E2 -8969.008} C_VEL
LIN {X 0,Y 440.616,Z 384.406,A -85,B 0,C 180,E1 -8969.972,E2 -8969.972} C_VEL
LIN {X 0,Y 440.931,Z 374.074,A -85,B 0,C 180,E1 -8970.748,E2 -8970.748} C_VEL
LIN {X 0,Y 441.197,Z 364.88,A -85,B 0,C 180,E1 -8971.273,E2 -8971.273} C_VEL
LIN {X 0,Y 441.434,Z 355.21,A -85,B 0,C 180,E1 -8971.681,E2 -8971.681} C_VEL
LIN {X 0,Y 441.558,Z 345.878,A -85,B 0,C 180,E1 -8971.949,E2 -8971.949} C_VEL
LIN {X 0,Y 442.11,Z 282.3,A -85,B 0,C 180,E1 -8973.069,E2 -8973.069} C_VEL
LIN {X 0,Y 439.708,Z 270.001,A -85,B 0,C 180,E1 -8973.389,E2 -8973.389} C_VEL
LIN {X 0,Y 439.596,Z 261.707,A -85,B 0,C 180,E1 -8975.187,E2 -8975.187} C_VEL
LIN {X 0,Y 439.39,Z 260.566,A -85,B 0,C 180,E1 -8975.485,E2 -8975.485} C_VEL
LIN {X 0,Y 439.403,Z 260.57,A -85,B 0,C 180,E1 -8978.417,E2 -8978.417} C_VEL
LIN {X 0,Y 439.417,Z 260.563,A -85,B 0,C 180,E1 -8981.345,E2 -8981.345} C_VEL
LIN {X 0,Y 439.451,Z 260.56,A -85,B 0,C 180,E1 -8984.225,E2 -8984.225} C_VEL
LIN {X 0,Y 439.474,Z 260.554,A -85,B 0,C 180,E1 -8988.002,E2 -8988.002} C_VEL
LIN {X 0,Y 439.538,Z 260.545,A -85,B 0,C 180,E1 -8991.727,E2 -8991.727} C_VEL
LIN {X 0,Y 439.614,Z 260.538,A -85,B 0,C 180,E1 -8994.497,E2 -8994.497} C_VEL
LIN {X 0,Y 439.627,Z 260.533,A -85,B 0,C 180,E1 -8998.169,E2 -8998.169} C_VEL
LIN {X 0,Y 439.754,Z 260.519,A -85,B 0,C 180,E1 -9000.001,E2 -9000.001} C_VEL
LIN {X 0,Y 439.648,Z 260.534,A -85,B 0,C 180,E1 -9002.75,E2 -9002.75} C_VEL
LIN {X 0,Y 439.609,Z 260.541,A -85,B 0,C 180,E1 -9006.426,E2 -9006.426} C_VEL
LIN {X 0,Y 439.492,Z 260.549,A -85,B 0,C 180,E1 -9009.202,E2 -9009.202} C_VEL
LIN {X 0,Y 439.457,Z 260.554,A -85,B 0,C 180,E1 -9012.939,E2 -9012.939} C_VEL
LIN {X 0,Y 439.44,Z 260.557,A -85,B 0,C 180,E1 -9016.35,E2 -9016.35} C_VEL
LIN {X 0,Y 439.395,Z 260.56,A -85,B 0,C 180,E1 -9019.627,E2 -9019.627} C_VEL
LIN {X 0,Y 439.358,Z 260.571,A -85,B 0,C 180,E1 -9022.576,E2 -9022.576} C_VEL
LIN {X 0,Y 439.399,Z 260.555,A -85,B 0,C 180,E1 -9025.586,E2 -9025.586} C_VEL
LIN {X 0,Y 439.419,Z 260.558,A -85,B 0,C 180,E1 -9028.674,E2 -9028.674} C_VEL
LIN {X 0,Y 439.368,Z 260.566,A -85,B 0,C 180,E1 -9031.861,E2 -9031.861} C_VEL
LIN {X 0,Y 439.396,Z 260.562,A -85,B 0,C 180,E1 -9035.157,E2 -9035.157} C_VEL
LIN {X 0,Y 439.393,Z 260.568,A -85,B 0,C 180,E1 -9038.594,E2 -9038.594} C_VEL
LIN {X 0,Y 439.394,Z 260.561,A -85,B 0,C 180,E1 -9041.259,E2 -9041.259} C_VEL
LIN {X 0,Y 439.397,Z 260.566,A -85,B 0,C 180,E1 -9044.73,E2 -9044.73} C_VEL
LIN {X 0,Y 439.393,Z 260.563,A -85,B 0,C 180,E1 -9047.797,E2 -9047.797} C_VEL
LIN {X 0,Y 439.434,Z 260.561,A -85,B 0,C 180,E1 -9050.229,E2 -9050.229} C_VEL
LIN {X 0,Y 439.374,Z 260.565,A -85,B 0,C 180,E1 -9053.714,E2 -9053.714} C_VEL
LIN {X 0,Y 439.371,Z 260.567,A -85,B 0,C 180,E1 -9057.055,E2 -9057.055} C_VEL
LIN {X 0,Y 439.381,Z 260.57,A -85,B 0,C 180,E1 -9060.275,E2 -9060.275} C_VEL
LIN {X 0,Y 439.427,Z 260.56,A -85,B 0,C 180,E1 -9063.397,E2 -9063.397} C_VEL
LIN {X 0,Y 439.462,Z 260.571,A -85,B 0,C 180,E1 -9064.99,E2 -9064.99} C_VEL
LIN {X 0,Y 440.878,Z 269.177,A -85,B 0,C 180,E1 -9066.764,E2 -9066.764} C_VEL
LIN {X 0,Y 440.329,Z 284.263,A -85,B 0,C 180,E1 -9069.688,E2 -9069.688} C_VEL
LIN {X 0,Y 439.627,Z 302.955,A -85,B 0,C 180,E1 -9073.277,E2 -9073.277} C_VEL
LIN {X 0,Y 439.275,Z 315.346,A -85,B 0,C 180,E1 -9075.641,E2 -9075.641} C_VEL
LIN {X 0,Y 441.812,Z 337.603,A -85,B 0,C 180,E1 -9076.129,E2 -9076.129} C_VEL
LIN {X 0,Y 441.31,Z 393.893,A -85,B 0,C 180,E1 -9077.118,E2 -9077.118} C_VEL
LIN {X 0,Y 441.047,Z 404.276,A -85,B 0,C 180,E1 -9077.432,E2 -9077.432} C_VEL
LIN {X 0,Y 440.633,Z 415.037,A -85,B 0,C 180,E1 -9077.917,E2 -9077.917} C_VEL
LIN {X 0,Y 440.164,Z 425.74,A -85,B 0,C 180,E1 -9078.604,E2 -9078.604} C_VEL
LIN {X 0,Y 439.748,Z 434.134,A -85,B 0,C 180,E1 -9079.293,E2 -9079.293} C_VEL
LIN {X 0,Y 439.39,Z 442.095,A -85,B 0,C 180,E1 -9080.1,E2 -9080.1} C_VEL
LIN {X 0,Y 439.067,Z 449.554,A -85,B 0,C 180,E1 -9081.022,E2 -9081.022} C_VEL
LIN {X 0,Y 438.75,Z 457.132,A -85,B 0,C 180,E1 -9082.175,E2 -9082.175} C_VEL
LIN {X 0,Y 438.556,Z 463.079,A -85,B 0,C 180,E1 -9083.328,E2 -9083.328} C_VEL
LIN {X 0,Y 438.428,Z 467.773,A -85,B 0,C 180,E1 -9084.481,E2 -9084.481} C_VEL
LIN {X 0,Y 438.374,Z 470.83,A -85,B 0,C 180,E1 -9085.403,E2 -9085.403} C_VEL
LIN {X 0,Y 438.352,Z 473.216,A -85,B 0,C 180,E1 -9086.323,E2 -9086.323} C_VEL
LIN {X 0,Y 438.401,Z 474.996,A -85,B 0,C 180,E1 -9087.244,E2 -9087.244} C_VEL
LIN {X 0,Y 438.344,Z 476.264,A -85,B 0,C 180,E1 -9088.163,E2 -9088.163} C_VEL
LIN {X 0,Y 438.339,Z 477.048,A -85,B 0,C 180,E1 -9089.082,E2 -9089.082} C_VEL
LIN {X 0,Y 438.348,Z 477.349,A -85,B 0,C 180,E1 -9090,E2 -9090} C_VEL
LIN {X 0,Y 438.352,Z 477.056,A -85,B 0,C 180,E1 -9090.919,E2 -9090.919} C_VEL
LIN {X 0,Y 438.344,Z 476.232,A -85,B 0,C 180,E1 -9091.838,E2 -9091.838} C_VEL
LIN {X 0,Y 438.403,Z 474.922,A -85,B 0,C 180,E1 -9092.757,E2 -9092.757} C_VEL
LIN {X 0,Y 438.34,Z 471.924,A -85,B 0,C 180,E1 -9094.138,E2 -9094.138} C_VEL
LIN {X 0,Y 438.428,Z 467.634,A -85,B 0,C 180,E1 -9095.519,E2 -9095.519} C_VEL
LIN {X 0,Y 438.597,Z 461.673,A -85,B 0,C 180,E1 -9096.903,E2 -9096.903} C_VEL
LIN {X 0,Y 438.746,Z 456.715,A -85,B 0,C 180,E1 -9097.826,E2 -9097.826} C_VEL
LIN {X 0,Y 438.966,Z 450.733,A -85,B 0,C 180,E1 -9098.749,E2 -9098.749} C_VEL
LIN {X 0,Y 439.308,Z 443.454,A -85,B 0,C 180,E1 -9099.67,E2 -9099.67} C_VEL
LIN {X 0,Y 439.618,Z 435.678,A -85,B 0,C 180,E1 -9100.477,E2 -9100.477} C_VEL
LIN {X 0,Y 439.996,Z 427.511,A -85,B 0,C 180,E1 -9101.167,E2 -9101.167} C_VEL
LIN {X 0,Y 440.309,Z 419.031,A -85,B 0,C 180,E1 -9101.742,E2 -9101.742} C_VEL
LIN {X 0,Y 440.698,Z 409.156,A -85,B 0,C 180,E1 -9102.257,E2 -9102.257} C_VEL
LIN {X 0,Y 441.103,Z 397.086,A -85,B 0,C 180,E1 -9102.684,E2 -9102.684} C_VEL
LIN {X 0,Y 441.33,Z 376.835,A -85,B 0,C 180,E1 -9103.065,E2 -9103.065} C_VEL
LIN {X 0,Y 441.534,Z 336.634,A -85,B 0,C 180,E1 -9103.753,E2 -9103.753} C_VEL
LIN {X 0,Y 439.284,Z 316.569,A -85,B 0,C 180,E1 -9104.181,E2 -9104.181} C_VEL
LIN {X 0,Y 439.914,Z 298.994,A -85,B 0,C 180,E1 -9107.67,E2 -9107.67} C_VEL
LIN {X 0,Y 440.646,Z 282.235,A -85,B 0,C 180,E1 -9111.03,E2 -9111.03} C_VEL
LIN {X 0,Y 441.202,Z 271.426,A -85,B 0,C 180,E1 -9113.219,E2 -9113.219} C_VEL
LIN {X 0,Y 439.548,Z 261.077,A -85,B 0,C 180,E1 -9115.449,E2 -9115.449} C_VEL
LIN {X 0,Y 439.44,Z 260.562,A -85,B 0,C 180,E1 -9115.582,E2 -9115.582} C_VEL
LIN {X 0,Y 439.418,Z 260.559,A -85,B 0,C 180,E1 -9118.673,E2 -9118.673} C_VEL
LIN {X 0,Y 439.37,Z 260.565,A -85,B 0,C 180,E1 -9122.03,E2 -9122.03} C_VEL
LIN {X 0,Y 439.394,Z 260.565,A -85,B 0,C 180,E1 -9125.34,E2 -9125.34} C_VEL
LIN {X 0,Y 439.384,Z 260.561,A -85,B 0,C 180,E1 -9128.594,E2 -9128.594} C_VEL
LIN {X 0,Y 439.388,Z 260.565,A -85,B 0,C 180,E1 -9131.256,E2 -9131.256} C_VEL
LIN {X 0,Y 439.4,Z 260.56,A -85,B 0,C 180,E1 -9134.729,E2 -9134.729} C_VEL
LIN {X 0,Y 439.394,Z 260.565,A -85,B 0,C 180,E1 -9137.795,E2 -9137.795} C_VEL
LIN {X 0,Y 439.392,Z 260.561,A -85,B 0,C 180,E1 -9140.223,E2 -9140.223} C_VEL
LIN {X 0,Y 439.372,Z 260.569,A -85,B 0,C 180,E1 -9143.712,E2 -9143.712} C_VEL
LIN {X 0,Y 439.369,Z 260.565,A -85,B 0,C 180,E1 -9147.053,E2 -9147.053} C_VEL
LIN {X 0,Y 439.379,Z 260.563,A -85,B 0,C 180,E1 -9150.273,E2 -9150.273} C_VEL
LIN {X 0,Y 439.427,Z 260.562,A -85,B 0,C 180,E1 -9153.396,E2 -9153.396} C_VEL
LIN {X 0,Y 439.383,Z 260.562,A -85,B 0,C 180,E1 -9156.429,E2 -9156.429} C_VEL
LIN {X 0,Y 439.384,Z 260.567,A -85,B 0,C 180,E1 -9159.396,E2 -9159.396} C_VEL
LIN {X 0,Y 439.427,Z 260.557,A -85,B 0,C 180,E1 -9162.309,E2 -9162.309} C_VEL
LIN {X 0,Y 439.443,Z 260.557,A -85,B 0,C 180,E1 -9165.173,E2 -9165.173} C_VEL
LIN {X 0,Y 439.478,Z 260.552,A -85,B 0,C 180,E1 -9168,E2 -9168} C_VEL
LIN {X 0,Y 439.543,Z 260.548,A -85,B 0,C 180,E1 -9171.725,E2 -9171.725} C_VEL
LIN {X 0,Y 439.615,Z 260.533,A -85,B 0,C 180,E1 -9174.495,E2 -9174.495} C_VEL
LIN {X 0,Y 439.63,Z 260.533,A -85,B 0,C 180,E1 -9178.167,E2 -9178.167} C_VEL
LIN {X 0,Y 439.757,Z 260.518,A -85,B 0,C 180,E1 -9179.999,E2 -9179.999} C_VEL
LIN {X 0,Y 439.65,Z 260.529,A -85,B 0,C 180,E1 -9182.748,E2 -9182.748} C_VEL
LIN {X 0,Y 439.611,Z 260.534,A -85,B 0,C 180,E1 -9186.424,E2 -9186.424} C_VEL
LIN {X 0,Y 439.494,Z 260.551,A -85,B 0,C 180,E1 -9189.201,E2 -9189.201} C_VEL
LIN {X 0,Y 439.497,Z 260.548,A -85,B 0,C 180,E1 -9192.726,E2 -9192.726} C_VEL
LIN {X 0,Y 439.44,Z 260.556,A -85,B 0,C 180,E1 -9196.348,E2 -9196.348} C_VEL
LIN {X 0,Y 439.423,Z 260.564,A -85,B 0,C 180,E1 -9199.624,E2 -9199.624} C_VEL
LIN {X 0,Y 439.356,Z 260.566,A -85,B 0,C 180,E1 -9202.575,E2 -9202.575} C_VEL
LIN {X 0,Y 439.398,Z 260.567,A -85,B 0,C 180,E1 -9205.584,E2 -9205.584} C_VEL
LIN {X 0,Y 439.409,Z 260.559,A -85,B 0,C 180,E1 -9208.673,E2 -9208.673} C_VEL
LIN {X 0,Y 439.362,Z 260.567,A -85,B 0,C 180,E1 -9212.03,E2 -9212.03} C_VEL
LIN {X 0,Y 439.387,Z 260.565,A -85,B 0,C 180,E1 -9215.34,E2 -9215.34} C_VEL
LIN {X 0,Y 439.389,Z 260.562,A -85,B 0,C 180,E1 -9218.593,E2 -9218.593} C_VEL
LIN {X 0,Y 439.39,Z 260.564,A -85,B 0,C 180,E1 -9221.258,E2 -9221.258} C_VEL
LIN {X 0,Y 439.397,Z 260.561,A -85,B 0,C 180,E1 -9224.728,E2 -9224.728} C_VEL
LIN {X 0,Y 439.403,Z 260.565,A -85,B 0,C 180,E1 -9227.797,E2 -9227.797} C_VEL
LIN {X 0,Y 439.44,Z 260.556,A -85,B 0,C 180,E1 -9230.229,E2 -9230.229} C_VEL
LIN {X 0,Y 439.367,Z 260.571,A -85,B 0,C 180,E1 -9233.713,E2 -9233.713} C_VEL
LIN {X 0,Y 439.363,Z 260.566,A -85,B 0,C 180,E1 -9237.054,E2 -9237.054} C_VEL
LIN {X 0,Y 439.373,Z 260.565,A -85,B 0,C 180,E1 -9240.274,E2 -9240.274} C_VEL
LIN {X 0,Y 439.419,Z 260.562,A -85,B 0,C 180,E1 -9243.396,E2 -9243.396} C_VEL
LIN {X 0,Y 439.379,Z 260.563,A -85,B 0,C 180,E1 -9246.429,E2 -9246.429} C_VEL
LIN {X 0,Y 439.384,Z 260.566,A -85,B 0,C 180,E1 -9249.397,E2 -9249.397} C_VEL
LIN {X 0,Y 439.423,Z 260.558,A -85,B 0,C 180,E1 -9252.309,E2 -9252.309} C_VEL
LIN {X 0,Y 439.439,Z 260.557,A -85,B 0,C 180,E1 -9255.174,E2 -9255.174} C_VEL
LIN {X 0,Y 439.475,Z 260.554,A -85,B 0,C 180,E1 -9258.001,E2 -9258.001} C_VEL
LIN {X 0,Y 439.539,Z 260.549,A -85,B 0,C 180,E1 -9261.726,E2 -9261.726} C_VEL
LIN {X 0,Y 439.607,Z 260.535,A -85,B 0,C 180,E1 -9264.495,E2 -9264.495} C_VEL
LIN {X 0,Y 439.624,Z 260.534,A -85,B 0,C 180,E1 -9268.168,E2 -9268.168} C_VEL
LIN {X 0,Y 439.753,Z 260.52,A -85,B 0,C 180,E1 -9270,E2 -9270} C_VEL
LIN {X 0,Y 439.612,Z 260.535,A -85,B 0,C 180,E1 -9270.998,E2 -9270.998} C_VEL
LIN {X 0,Y 438.896,Z 260.629,A -85,B 0,C 180,E1 -9271.763,E2 -9271.763} C_VEL
LIN {X 0,Y 435.916,Z 260.995,A -85,B 0,C 180,E1 -9273.002,E2 -9273.002} C_VEL
LIN {X 0,Y 433.463,Z 261.303,A -85,B 0,C 180,E1 -9274.002,E2 -9274.002} C_VEL
LIN {X 0,Y 432.489,Z 261.422,A -85,B 0,C 180,E1 -9274.777,E2 -9274.777} C_VEL
LIN {X 0,Y 432.452,Z 261.427,A -85,B 0,C 180,E1 -9275.039,E2 -9275.039} C_VEL
LIN {X 0,Y 432.551,Z 261.42,A -85,B 0,C 180,E1 -9277.653,E2 -9277.653} C_VEL
LIN {X 0,Y 432.397,Z 261.435,A -85,B 0,C 180,E1 -9281.247,E2 -9281.247} C_VEL
LIN {X 0,Y 432.422,Z 261.431,A -85,B 0,C 180,E1 -9283.152,E2 -9283.152} C_VEL
LIN {X 0,Y 432.402,Z 261.433,A -85,B 0,C 180,E1 -9286.479,E2 -9286.479} C_VEL
LIN {X 0,Y 432.328,Z 261.445,A -85,B 0,C 180,E1 -9289.96,E2 -9289.96} C_VEL
LIN {X 0,Y 432.306,Z 261.445,A -85,B 0,C 180,E1 -9292.964,E2 -9292.964} C_VEL
LIN {X 0,Y 432.339,Z 261.443,A -85,B 0,C 180,E1 -9296.033,E2 -9296.033} C_VEL
LIN {X 0,Y 432.331,Z 261.443,A -85,B 0,C 180,E1 -9299.187,E2 -9299.187} C_VEL
LIN {X 0,Y 432.417,Z 261.638,A -85,B 0,C 180,E1 -9302.434,E2 -9302.434} C_VEL
LIN {X 0,Y 432.584,Z 266.825,A -85,B 0,C 180,E1 -9303.783,E2 -9303.783} C_VEL
LIN {X 0,Y 432.498,Z 270.401,A -85,B 0,C 180,E1 -9304.697,E2 -9304.697} C_VEL
LIN {X 0,Y 434.984,Z 284.444,A -85,B 0,C 180,E1 -9305.034,E2 -9305.034} C_VEL
LIN {X 0,Y 434.375,Z 346.001,A -85,B 0,C 180,E1 -9306.121,E2 -9306.121} C_VEL
LIN {X 0,Y 434.139,Z 355.483,A -85,B 0,C 180,E1 -9306.398,E2 -9306.398} C_VEL
LIN {X 0,Y 433.934,Z 365.103,A -85,B 0,C 180,E1 -9306.815,E2 -9306.815} C_VEL
LIN {X 0,Y 433.614,Z 375.43,A -85,B 0,C 180,E1 -9307.423,E2 -9307.423} C_VEL
LIN {X 0,Y 433.318,Z 385.079,A -85,B 0,C 180,E1 -9308.189,E2 -9308.189} C_VEL
LIN {X 0,Y 432.963,Z 393.438,A -85,B 0,C 180,E1 -9309.026,E2 -9309.026} C_VEL
LIN {X 0,Y 432.572,Z 400.747,A -85,B 0,C 180,E1 -9309.922,E2 -9309.922} C_VEL
LIN {X 0,Y 432.316,Z 406.706,A -85,B 0,C 180,E1 -9310.805,E2 -9310.805} C_VEL
LIN {X 0,Y 432.029,Z 412.441,A -85,B 0,C 180,E1 -9311.832,E2 -9311.832} C_VEL
LIN {X 0,Y 431.824,Z 417.36,A -85,B 0,C 180,E1 -9312.915,E2 -9312.915} C_VEL
LIN {X 0,Y 431.6,Z 422.082,A -85,B 0,C 180,E1 -9314.237,E2 -9314.237} C_VEL
LIN {X 0,Y 431.398,Z 425.99,A -85,B 0,C 180,E1 -9315.79,E2 -9315.79} C_VEL
LIN {X 0,Y 431.257,Z 428.13,A -85,B 0,C 180,E1 -9317.166,E2 -9317.166} C_VEL
LIN {X 0,Y 431.187,Z 429.187,A -85,B 0,C 180,E1 -9318.568,E2 -9318.568} C_VEL
LIN {X 0,Y 431.222,Z 429.121,A -85,B 0,C 180,E1 -9319.994,E2 -9319.994} C_VEL
LIN {X 0,Y 431.321,Z 427.862,A -85,B 0,C 180,E1 -9321.453,E2 -9321.453} C_VEL
LIN {X 0,Y 431.509,Z 425.147,A -85,B 0,C 180,E1 -9322.944,E2 -9322.944} C_VEL
LIN {X 0,Y 431.765,Z 420.88,A -85,B 0,C 180,E1 -9324.474,E2 -9324.474} C_VEL
LIN {X 0,Y 432.032,Z 416.227,A -85,B 0,C 180,E1 -9325.705,E2 -9325.705} C_VEL
LIN {X 0,Y 432.341,Z 409.883,A -85,B 0,C 180,E1 -9327.006,E2 -9327.006} C_VEL
LIN {X 0,Y 432.721,Z 402.709,A -85,B 0,C 180,E1 -9328.141,E2 -9328.141} C_VEL
LIN {X 0,Y 433.156,Z 395.701,A -85,B 0,C 180,E1 -9329.044,E2 -9329.044} C_VEL
LIN {X 0,Y 433.492,Z 388.322,A -85,B 0,C 180,E1 -9329.83,E2 -9329.83} C_VEL
LIN {X 0,Y 433.853,Z 380.314,A -85,B 0,C 180,E1 -9330.526,E2 -9330.526} C_VEL
LIN {X 0,Y 434.119,Z 371.513,A -85,B 0,C 180,E1 -9331.14,E2 -9331.14} C_VEL
LIN {X 0,Y 434.492,Z 360.951,A -85,B 0,C 180,E1 -9331.698,E2 -9331.698} C_VEL
LIN {X 0,Y 434.656,Z 349.323,A -85,B 0,C 180,E1 -9332.104,E2 -9332.104} C_VEL
LIN {X 0,Y 434.918,Z 326.973,A -85,B 0,C 180,E1 -9332.531,E2 -9332.531} C_VEL
LIN {X 0,Y 435.39,Z 283.707,A -85,B 0,C 180,E1 -9333.297,E2 -9333.297} C_VEL
LIN {X 0,Y 432.743,Z 270.343,A -85,B 0,C 180,E1 -9333.659,E2 -9333.659} C_VEL
LIN {X 0,Y 432.789,Z 264.068,A -85,B 0,C 180,E1 -9335.027,E2 -9335.027} C_VEL
LIN {X 0,Y 432.358,Z 261.442,A -85,B 0,C 180,E1 -9335.643,E2 -9335.643} C_VEL
LIN {X 0,Y 432.339,Z 261.448,A -85,B 0,C 180,E1 -9339.047,E2 -9339.047} C_VEL
LIN {X 0,Y 432.367,Z 261.444,A -85,B 0,C 180,E1 -9342.012,E2 -9342.012} C_VEL
LIN {X 0,Y 432.384,Z 261.438,A -85,B 0,C 180,E1 -9344.927,E2 -9344.927} C_VEL
LIN {X 0,Y 432.449,Z 261.428,A -85,B 0,C 180,E1 -9347.804,E2 -9347.804} C_VEL
LIN {X 0,Y 432.482,Z 261.424,A -85,B 0,C 180,E1 -9351.591,E2 -9351.591} C_VEL
LIN {X 0,Y 432.59,Z 261.414,A -85,B 0,C 180,E1 -9354.407,E2 -9354.407} C_VEL
LIN {X 0,Y 432.597,Z 261.409,A -85,B 0,C 180,E1 -9358.139,E2 -9358.139} C_VEL
LIN {X 0,Y 432.724,Z 261.395,A -85,B 0,C 180,E1 -9360.001,E2 -9360.001} C_VEL
LIN {X 0,Y 432.597,Z 261.411,A -85,B 0,C 180,E1 -9362.794,E2 -9362.794} C_VEL
LIN {X 0,Y 432.564,Z 261.418,A -85,B 0,C 180,E1 -9366.531,E2 -9366.531} C_VEL
LIN {X 0,Y 432.435,Z 261.427,A -85,B 0,C 180,E1 -9369.354,E2 -9369.354} C_VEL
LIN {X 0,Y 432.423,Z 261.431,A -85,B 0,C 180,E1 -9372.804,E2 -9372.804} C_VEL
LIN {X 0,Y 432.405,Z 261.432,A -85,B 0,C 180,E1 -9376.48,E2 -9376.48} C_VEL
LIN {X 0,Y 432.332,Z 261.442,A -85,B 0,C 180,E1 -9379.961,E2 -9379.961} C_VEL
LIN {X 0,Y 432.312,Z 261.445,A -85,B 0,C 180,E1 -9382.965,E2 -9382.965} C_VEL
LIN {X 0,Y 432.358,Z 261.435,A -85,B 0,C 180,E1 -9386.033,E2 -9386.033} C_VEL
LIN {X 0,Y 432.346,Z 261.434,A -85,B 0,C 180,E1 -9389.188,E2 -9389.188} C_VEL
LIN {X 0,Y 432.32,Z 261.448,A -85,B 0,C 180,E1 -9392.294,E2 -9392.294} C_VEL
LIN {X 0,Y 432.336,Z 261.446,A -85,B 0,C 180,E1 -9394.678,E2 -9394.678} C_VEL
LIN {X 0,Y 432.348,Z 261.439,A -85,B 0,C 180,E1 -9398.149,E2 -9398.149} C_VEL
LIN {X 0,Y 432.363,Z 261.437,A -85,B 0,C 180,E1 -9401.608,E2 -9401.608} C_VEL
LIN {X 0,Y 432.33,Z 261.444,A -85,B 0,C 180,E1 -9404.348,E2 -9404.348} C_VEL
LIN {X 0,Y 432.317,Z 261.445,A -85,B 0,C 180,E1 -9407.017,E2 -9407.017} C_VEL
LIN {X 0,Y 432.338,Z 261.442,A -85,B 0,C 180,E1 -9409.821,E2 -9409.821} C_VEL
LIN {X 0,Y 432.313,Z 261.446,A -85,B 0,C 180,E1 -9413.024,E2 -9413.024} C_VEL
LIN {X 0,Y 432.358,Z 261.441,A -85,B 0,C 180,E1 -9415.997,E2 -9415.997} C_VEL
LIN {X 0,Y 432.346,Z 261.443,A -85,B 0,C 180,E1 -9419.491,E2 -9419.491} C_VEL
LIN {X 0,Y 432.39,Z 261.44,A -85,B 0,C 180,E1 -9422.929,E2 -9422.929} C_VEL
LIN {X 0,Y 432.401,Z 261.464,A -85,B 0,C 180,E1 -9424.81,E2 -9424.81} C_VEL
LIN {X 0,Y 433.897,Z 270.072,A -85,B 0,C 180,E1 -9426.62,E2 -9426.62} C_VEL
LIN {X 0,Y 433.438,Z 281.393,A -85,B 0,C 180,E1 -9428.853,E2 -9428.853} C_VEL
LIN {X 0,Y 432.819,Z 297.64,A -85,B 0,C 180,E1 -9432.031,E2 -9432.031} C_VEL
LIN {X 0,Y 432.251,Z 314.856,A -85,B 0,C 180,E1 -9435.369,E2 -9435.369} C_VEL
LIN {X 0,Y 434.945,Z 337.676,A -85,B 0,C 180,E1 -9435.891,E2 -9435.891} C_VEL
LIN {X 0,Y 434.444,Z 393.306,A -85,B 0,C 180,E1 -9436.893,E2 -9436.893} C_VEL
LIN {X 0,Y 434.157,Z 403.397,A -85,B 0,C 180,E1 -9437.199,E2 -9437.199} C_VEL
LIN {X 0,Y 433.7,Z 414.83,A -85,B 0,C 180,E1 -9437.721,E2 -9437.721} C_VEL
LIN {X 0,Y 433.207,Z 425.478,A -85,B 0,C 180,E1 -9438.419,E2 -9438.419} C_VEL
LIN {X 0,Y 432.748,Z 433.847,A -85,B 0,C 180,E1 -9439.118,E2 -9439.118} C_VEL
LIN {X 0,Y 432.39,Z 441.793,A -85,B 0,C 180,E1 -9439.938,E2 -9439.938} C_VEL
LIN {X 0,Y 432.04,Z 449.237,A -85,B 0,C 180,E1 -9440.875,E2 -9440.875} C_VEL
LIN {X 0,Y 431.682,Z 456.8,A -85,B 0,C 180,E1 -9442.046,E2 -9442.046} C_VEL
LIN {X 0,Y 431.487,Z 462.729,A -85,B 0,C 180,E1 -9443.219,E2 -9443.219} C_VEL
LIN {X 0,Y 431.329,Z 467.415,A -85,B 0,C 180,E1 -9444.39,E2 -9444.39} C_VEL
LIN {X 0,Y 431.306,Z 470.468,A -85,B 0,C 180,E1 -9445.327,E2 -9445.327} C_VEL
LIN {X 0,Y 431.252,Z 472.853,A -85,B 0,C 180,E1 -9446.263,E2 -9446.263} C_VEL
LIN {X 0,Y 431.327,Z 474.627,A -85,B 0,C 180,E1 -9447.198,E2 -9447.198} C_VEL
LIN {X 0,Y 431.265,Z 475.884,A -85,B 0,C 180,E1 -9448.133,E2 -9448.133} C_VEL
LIN {X 0,Y 431.251,Z 476.658,A -85,B 0,C 180,E1 -9449.066,E2 -9449.066} C_VEL
LIN {X 0,Y 431.287,Z 476.953,A -85,B 0,C 180,E1 -9450,E2 -9450} C_VEL
LIN {X 0,Y 431.263,Z 476.657,A -85,B 0,C 180,E1 -9450.934,E2 -9450.934} C_VEL
LIN {X 0,Y 431.265,Z 475.82,A -85,B 0,C 180,E1 -9451.868,E2 -9451.868} C_VEL
LIN {X 0,Y 431.33,Z 474.496,A -85,B 0,C 180,E1 -9452.802,E2 -9452.802} C_VEL
LIN {X 0,Y 431.256,Z 471.482,A -85,B 0,C 180,E1 -9454.206,E2 -9454.206} C_VEL
LIN {X 0,Y 431.329,Z 467.168,A -85,B 0,C 180,E1 -9455.61,E2 -9455.61} C_VEL
LIN {X 0,Y 431.53,Z 461.17,A -85,B 0,C 180,E1 -9457.016,E2 -9457.016} C_VEL
LIN {X 0,Y 431.679,Z 456.184,A -85,B 0,C 180,E1 -9457.954,E2 -9457.954} C_VEL
LIN {X 0,Y 431.935,Z 450.174,A -85,B 0,C 180,E1 -9458.892,E2 -9458.892} C_VEL
LIN {X 0,Y 432.281,Z 442.857,A -85,B 0,C 180,E1 -9459.829,E2 -9459.829} C_VEL
LIN {X 0,Y 432.601,Z 435.036,A -85,B 0,C 180,E1 -9460.649,E2 -9460.649} C_VEL
LIN {X 0,Y 433.01,Z 426.813,A -85,B 0,C 180,E1 -9461.35,E2 -9461.35} C_VEL
LIN {X 0,Y 433.334,Z 418.256,A -85,B 0,C 180,E1 -9461.934,E2 -9461.934} C_VEL
LIN {X 0,Y 433.814,Z 407.029,A -85,B 0,C 180,E1 -9462.514,E2 -9462.514} C_VEL
LIN {X 0,Y 434.126,Z 395.645,A -85,B 0,C 180,E1 -9462.891,E2 -9462.891} C_VEL
LIN {X 0,Y 434.451,Z 370.868,A -85,B 0,C 180,E1 -9463.35,E2 -9463.35} C_VEL
LIN {X 0,Y 434.6,Z 337.074,A -85,B 0,C 180,E1 -9463.941,E2 -9463.941} C_VEL
LIN {X 0,Y 432.237,Z 316.274,A -85,B 0,C 180,E1 -9464.387,E2 -9464.387} C_VEL
LIN {X 0,Y 432.952,Z 298.537,A -85,B 0,C 180,E1 -9467.964,E2 -9467.964} C_VEL
LIN {X 0,Y 433.638,Z 282.987,A -85,B 0,C 180,E1 -9471.137,E2 -9471.137} C_VEL
LIN {X 0,Y 434.211,Z 272.194,A -85,B 0,C 180,E1 -9473.362,E2 -9473.362} C_VEL
LIN {X 0,Y 432.399,Z 261.439,A -85,B 0,C 180,E1 -9475.739,E2 -9475.739} C_VEL
LIN {X 0,Y 432.343,Z 261.444,A -85,B 0,C 180,E1 -9479.187,E2 -9479.187} C_VEL
LIN {X 0,Y 432.323,Z 261.441,A -85,B 0,C 180,E1 -9482.442,E2 -9482.442} C_VEL
LIN {X 0,Y 432.344,Z 261.445,A -85,B 0,C 180,E1 -9485.631,E2 -9485.631} C_VEL
LIN {X 0,Y 432.354,Z 261.442,A -85,B 0,C 180,E1 -9489.342,E2 -9489.342} C_VEL
LIN {X 0,Y 432.333,Z 261.444,A -85,B 0,C 180,E1 -9491.796,E2 -9491.796} C_VEL
LIN {X 0,Y 432.333,Z 261.44,A -85,B 0,C 180,E1 -9494.347,E2 -9494.347} C_VEL
LIN {X 0,Y 432.318,Z 261.443,A -85,B 0,C 180,E1 -9497.015,E2 -9497.015} C_VEL
LIN {X 0,Y 432.332,Z 261.444,A -85,B 0,C 180,E1 -9499.82,E2 -9499.82} C_VEL
LIN {X 0,Y 432.304,Z 261.445,A -85,B 0,C 180,E1 -9503.021,E2 -9503.021} C_VEL
LIN {X 0,Y 432.357,Z 261.439,A -85,B 0,C 180,E1 -9505.996,E2 -9505.996} C_VEL
LIN {X 0,Y 432.344,Z 261.445,A -85,B 0,C 180,E1 -9509.489,E2 -9509.489} C_VEL
LIN {X 0,Y 432.39,Z 261.434,A -85,B 0,C 180,E1 -9512.928,E2 -9512.928} C_VEL
LIN {X 0,Y 432.368,Z 261.438,A -85,B 0,C 180,E1 -9516.023,E2 -9516.023} C_VEL
LIN {X 0,Y 432.346,Z 261.44,A -85,B 0,C 180,E1 -9519.045,E2 -9519.045} C_VEL
LIN {X 0,Y 432.373,Z 261.437,A -85,B 0,C 180,E1 -9522.01,E2 -9522.01} C_VEL
LIN {X 0,Y 432.39,Z 261.434,A -85,B 0,C 180,E1 -9524.926,E2 -9524.926} C_VEL
LIN {X 0,Y 432.454,Z 261.43,A -85,B 0,C 180,E1 -9527.803,E2 -9527.803} C_VEL
LIN {X 0,Y 432.487,Z 261.429,A -85,B 0,C 180,E1 -9531.59,E2 -9531.59} C_VEL
LIN {X 0,Y 432.592,Z 261.408,A -85,B 0,C 180,E1 -9534.405,E2 -9534.405} C_VEL
LIN {X 0,Y 432.6,Z 261.408,A -85,B 0,C 180,E1 -9538.137,E2 -9538.137} C_VEL
LIN {X 0,Y 432.727,Z 261.394,A -85,B 0,C 180,E1 -9539.999,E2 -9539.999} C_VEL
LIN {X 0,Y 432.6,Z 261.407,A -85,B 0,C 180,E1 -9542.793,E2 -9542.793} C_VEL
LIN {X 0,Y 432.566,Z 261.411,A -85,B 0,C 180,E1 -9546.53,E2 -9546.53} C_VEL
LIN {X 0,Y 432.437,Z 261.432,A -85,B 0,C 180,E1 -9549.352,E2 -9549.352} C_VEL
LIN {X 0,Y 432.437,Z 261.428,A -85,B 0,C 180,E1 -9552.811,E2 -9552.811} C_VEL
LIN {X 0,Y 432.405,Z 261.432,A -85,B 0,C 180,E1 -9556.478,E2 -9556.478} C_VEL
LIN {X 0,Y 432.365,Z 261.439,A -85,B 0,C 180,E1 -9559.958,E2 -9559.958} C_VEL
LIN {X 0,Y 432.311,Z 261.444,A -85,B 0,C 180,E1 -9562.964,E2 -9562.964} C_VEL
LIN {X 0,Y 432.356,Z 261.44,A -85,B 0,C 180,E1 -9566.032,E2 -9566.032} C_VEL
LIN {X 0,Y 432.334,Z 261.443,A -85,B 0,C 180,E1 -9569.187,E2 -9569.187} C_VEL
LIN {X 0,Y 432.314,Z 261.443,A -85,B 0,C 180,E1 -9572.442,E2 -9572.442} C_VEL
LIN {X 0,Y 432.337,Z 261.447,A -85,B 0,C 180,E1 -9575.632,E2 -9575.632} C_VEL
LIN {X 0,Y 432.351,Z 261.439,A -85,B 0,C 180,E1 -9578.717,E2 -9578.717} C_VEL
LIN {X 0,Y 432.357,Z 261.443,A -85,B 0,C 180,E1 -9581.793,E2 -9581.793} C_VEL
LIN {X 0,Y 432.369,Z 261.443,A -85,B 0,C 180,E1 -9585.658,E2 -9585.658} C_VEL
LIN {X 0,Y 432.364,Z 261.437,A -85,B 0,C 180,E1 -9588.392,E2 -9588.392} C_VEL
LIN {X 0,Y 432.341,Z 261.444,A -85,B 0,C 180,E1 -9591.851,E2 -9591.851} C_VEL
LIN {X 0,Y 432.331,Z 261.444,A -85,B 0,C 180,E1 -9595.323,E2 -9595.323} C_VEL
LIN {X 0,Y 432.312,Z 261.444,A -85,B 0,C 180,E1 -9598.654,E2 -9598.654} C_VEL
LIN {X 0,Y 432.372,Z 261.44,A -85,B 0,C 180,E1 -9601.876,E2 -9601.876} C_VEL
LIN {X 0,Y 432.343,Z 261.44,A -85,B 0,C 180,E1 -9604.999,E2 -9604.999} C_VEL
LIN {X 0,Y 432.351,Z 261.441,A -85,B 0,C 180,E1 -9608.046,E2 -9608.046} C_VEL
LIN {X 0,Y 432.378,Z 261.436,A -85,B 0,C 180,E1 -9611.029,E2 -9611.029} C_VEL
LIN {X 0,Y 432.422,Z 261.433,A -85,B 0,C 180,E1 -9613.961,E2 -9613.961} C_VEL
LIN {X 0,Y 432.451,Z 261.431,A -85,B 0,C 180,E1 -9617.803,E2 -9617.803} C_VEL
LIN {X 0,Y 432.483,Z 261.428,A -85,B 0,C 180,E1 -9621.59,E2 -9621.59} C_VEL
LIN {X 0,Y 432.584,Z 261.41,A -85,B 0,C 180,E1 -9624.406,E2 -9624.406} C_VEL
LIN {X 0,Y 432.593,Z 261.41,A -85,B 0,C 180,E1 -9628.138,E2 -9628.138} C_VEL
LIN {X 0,Y 432.723,Z 261.395,A -85,B 0,C 180,E1 -9630,E2 -9630} C_VEL
LIN {X 0,Y 432.583,Z 261.41,A -85,B 0,C 180,E1 -9632.793,E2 -9632.793} C_VEL
LIN {X 0,Y 432.452,Z 261.427,A -85,B 0,C 180,E1 -9635.039,E2 -9635.039} C_VEL
LIN {X 0,Y 431.892,Z 261.501,A -85,B 0,C 180,E1 -9635.817,E2 -9635.817} C_VEL
LIN {X 0,Y 429.046,Z 261.851,A -85,B 0,C 180,E1 -9637.081,E2 -9637.081} C_VEL
LIN {X 0,Y 426.564,Z 262.162,A -85,B 0,C 180,E1 -9638.102,E2 -9638.102} C_VEL
LIN {X 0,Y 425.484,Z 262.295,A -85,B 0,C 180,E1 -9638.891,E2 -9638.891} C_VEL
LIN {X 0,Y 425.393,Z 262.307,A -85,B 0,C 180,E1 -9639.159,E2 -9639.159} C_VEL
LIN {X 0,Y 425.394,Z 262.306,A -85,B 0,C 180,E1 -9642.91,E2 -9642.91} C_VEL
LIN {X 0,Y 425.351,Z 262.311,A -85,B 0,C 180,E1 -9646.605,E2 -9646.605} C_VEL
LIN {X 0,Y 425.318,Z 262.32,A -85,B 0,C 180,E1 -9649.635,E2 -9649.635} C_VEL
LIN {X 0,Y 425.293,Z 262.321,A -85,B 0,C 180,E1 -9653.365,E2 -9653.365} C_VEL
LIN {X 0,Y 425.329,Z 262.314,A -85,B 0,C 180,E1 -9656.842,E2 -9656.842} C_VEL
LIN {X 0,Y 425.278,Z 262.326,A -85,B 0,C 180,E1 -9659.72,E2 -9659.72} C_VEL
LIN {X 0,Y 425.326,Z 262.323,A -85,B 0,C 180,E1 -9662.275,E2 -9662.275} C_VEL
LIN {X 0,Y 425.589,Z 267.268,A -85,B 0,C 180,E1 -9663.586,E2 -9663.586} C_VEL
LIN {X 0,Y 425.488,Z 270.733,A -85,B 0,C 180,E1 -9664.478,E2 -9664.478} C_VEL
LIN {X 0,Y 428.063,Z 285.008,A -85,B 0,C 180,E1 -9664.827,E2 -9664.827} C_VEL
LIN {X 0,Y 427.406,Z 347.143,A -85,B 0,C 180,E1 -9665.949,E2 -9665.949} C_VEL
LIN {X 0,Y 427.163,Z 357.627,A -85,B 0,C 180,E1 -9666.278,E2 -9666.278} C_VEL
LIN {X 0,Y 426.941,Z 369.472,A -85,B 0,C 180,E1 -9666.855,E2 -9666.855} C_VEL
LIN {X 0,Y 426.548,Z 378.849,A -85,B 0,C 180,E1 -9667.487,E2 -9667.487} C_VEL
LIN {X 0,Y 426.259,Z 387.447,A -85,B 0,C 180,E1 -9668.225,E2 -9668.225} C_VEL
LIN {X 0,Y 425.91,Z 394.672,A -85,B 0,C 180,E1 -9668.982,E2 -9668.982} C_VEL
LIN {X 0,Y 425.529,Z 401.519,A -85,B 0,C 180,E1 -9669.848,E2 -9669.848} C_VEL
LIN {X 0,Y 425.284,Z 407.082,A -85,B 0,C 180,E1 -9670.69,E2 -9670.69} C_VEL
LIN {X 0,Y 425.021,Z 412.412,A -85,B 0,C 180,E1 -9671.652,E2 -9671.652} C_VEL
LIN {X 0,Y 424.786,Z 417.246,A -85,B 0,C 180,E1 -9672.712,E2 -9672.712} C_VEL
LIN {X 0,Y 424.591,Z 420.68,A -85,B 0,C 180,E1 -9673.626,E2 -9673.626} C_VEL
LIN {X 0,Y 424.476,Z 423.696,A -85,B 0,C 180,E1 -9674.608,E2 -9674.608} C_VEL
LIN {X 0,Y 424.287,Z 426.662,A -85,B 0,C 180,E1 -9675.919,E2 -9675.919} C_VEL
LIN {X 0,Y 424.164,Z 428.583,A -85,B 0,C 180,E1 -9677.21,E2 -9677.21} C_VEL
LIN {X 0,Y 424.12,Z 429.546,A -85,B 0,C 180,E1 -9678.485,E2 -9678.485} C_VEL
LIN {X 0,Y 424.151,Z 429.603,A -85,B 0,C 180,E1 -9679.745,E2 -9679.745} C_VEL
LIN {X 0,Y 424.202,Z 428.643,A -85,B 0,C 180,E1 -9681.138,E2 -9681.138} C_VEL
LIN {X 0,Y 424.413,Z 426.404,A -85,B 0,C 180,E1 -9682.639,E2 -9682.639} C_VEL
LIN {X 0,Y 424.656,Z 422.536,A -85,B 0,C 180,E1 -9684.186,E2 -9684.186} C_VEL
LIN {X 0,Y 424.892,Z 419.137,A -85,B 0,C 180,E1 -9685.206,E2 -9685.206} C_VEL
LIN {X 0,Y 425.16,Z 414.196,A -85,B 0,C 180,E1 -9686.376,E2 -9686.376} C_VEL
LIN {X 0,Y 425.433,Z 408.842,A -85,B 0,C 180,E1 -9687.403,E2 -9687.403} C_VEL
LIN {X 0,Y 425.768,Z 402.742,A -85,B 0,C 180,E1 -9688.365,E2 -9688.365} C_VEL
LIN {X 0,Y 426.2,Z 395.865,A -85,B 0,C 180,E1 -9689.258,E2 -9689.258} C_VEL
LIN {X 0,Y 426.555,Z 389.306,A -85,B 0,C 180,E1 -9689.971,E2 -9689.971} C_VEL
LIN {X 0,Y 426.883,Z 382.169,A -85,B 0,C 180,E1 -9690.619,E2 -9690.619} C_VEL
LIN {X 0,Y 427.202,Z 373.292,A -85,B 0,C 180,E1 -9691.27,E2 -9691.27} C_VEL
LIN {X 0,Y 427.519,Z 364.068,A -85,B 0,C 180,E1 -9691.791,E2 -9691.791} C_VEL
LIN {X 0,Y 427.738,Z 353.441,A -85,B 0,C 180,E1 -9692.228,E2 -9692.228} C_VEL
LIN {X 0,Y 427.909,Z 338.365,A -85,B 0,C 180,E1 -9692.578,E2 -9692.578} C_VEL
LIN {X 0,Y 428.518,Z 284.431,A -85,B 0,C 180,E1 -9693.548,E2 -9693.548} C_VEL
LIN {X 0,Y 425.806,Z 270.734,A -85,B 0,C 180,E1 -9693.932,E2 -9693.932} C_VEL
LIN {X 0,Y 425.804,Z 265.048,A -85,B 0,C 180,E1 -9695.198,E2 -9695.198} C_VEL
LIN {X 0,Y 425.308,Z 262.321,A -85,B 0,C 180,E1 -9695.86,E2 -9695.86} C_VEL
LIN {X 0,Y 425.281,Z 262.329,A -85,B 0,C 180,E1 -9698.682,E2 -9698.682} C_VEL
LIN {X 0,Y 425.322,Z 262.32,A -85,B 0,C 180,E1 -9701.703,E2 -9701.703} C_VEL
LIN {X 0,Y 425.337,Z 262.318,A -85,B 0,C 180,E1 -9704.671,E2 -9704.671} C_VEL
LIN {X 0,Y 425.402,Z 262.305,A -85,B 0,C 180,E1 -9707.599,E2 -9707.599} C_VEL
LIN {X 0,Y 425.433,Z 262.302,A -85,B 0,C 180,E1 -9711.451,E2 -9711.451} C_VEL
LIN {X 0,Y 425.566,Z 262.289,A -85,B 0,C 180,E1 -9714.314,E2 -9714.314} C_VEL
LIN {X 0,Y 425.566,Z 262.284,A -85,B 0,C 180,E1 -9718.108,E2 -9718.108} C_VEL
LIN {X 0,Y 425.693,Z 262.271,A -85,B 0,C 180,E1 -9720.001,E2 -9720.001} C_VEL
LIN {X 0,Y 425.549,Z 262.289,A -85,B 0,C 180,E1 -9722.841,E2 -9722.841} C_VEL
LIN {X 0,Y 425.522,Z 262.294,A -85,B 0,C 180,E1 -9726.64,E2 -9726.64} C_VEL
LIN {X 0,Y 425.393,Z 262.305,A -85,B 0,C 180,E1 -9729.51,E2 -9729.51} C_VEL
LIN {X 0,Y 425.385,Z 262.308,A -85,B 0,C 180,E1 -9732.905,E2 -9732.905} C_VEL
LIN {X 0,Y 425.354,Z 262.309,A -85,B 0,C 180,E1 -9736.606,E2 -9736.606} C_VEL
LIN {X 0,Y 425.321,Z 262.313,A -85,B 0,C 180,E1 -9739.637,E2 -9739.637} C_VEL
LIN {X 0,Y 425.3,Z 262.316,A -85,B 0,C 180,E1 -9743.366,E2 -9743.366} C_VEL
LIN {X 0,Y 425.345,Z 262.315,A -85,B 0,C 180,E1 -9746.846,E2 -9746.846} C_VEL
LIN {X 0,Y 425.312,Z 262.31,A -85,B 0,C 180,E1 -9749.718,E2 -9749.718} C_VEL
LIN {X 0,Y 425.277,Z 262.316,A -85,B 0,C 180,E1 -9753.049,E2 -9753.049} C_VEL
LIN {X 0,Y 425.28,Z 262.321,A -85,B 0,C 180,E1 -9755.93,E2 -9755.93} C_VEL
LIN {X 0,Y 425.308,Z 262.318,A -85,B 0,C 180,E1 -9759.047,E2 -9759.047} C_VEL
LIN {X 0,Y 425.311,Z 262.317,A -85,B 0,C 180,E1 -9761.963,E2 -9761.963} C_VEL
LIN {X 0,Y 425.281,Z 262.32,A -85,B 0,C 180,E1 -9765.284,E2 -9765.284} C_VEL
LIN {X 0,Y 425.272,Z 262.324,A -85,B 0,C 180,E1 -9768.622,E2 -9768.622} C_VEL
LIN {X 0,Y 425.313,Z 262.317,A -85,B 0,C 180,E1 -9771.104,E2 -9771.104} C_VEL
LIN {X 0,Y 425.298,Z 262.323,A -85,B 0,C 180,E1 -9774.665,E2 -9774.665} C_VEL
LIN {X 0,Y 425.264,Z 262.326,A -85,B 0,C 180,E1 -9778.074,E2 -9778.074} C_VEL
LIN {X 0,Y 425.33,Z 262.318,A -85,B 0,C 180,E1 -9781.369,E2 -9781.369} C_VEL
LIN {X 0,Y 425.354,Z 262.362,A -85,B 0,C 180,E1 -9784.61,E2 -9784.61} C_VEL
LIN {X 0,Y 426.896,Z 271.01,A -85,B 0,C 180,E1 -9786.471,E2 -9786.471} C_VEL
LIN {X 0,Y 426.461,Z 282.336,A -85,B 0,C 180,E1 -9788.743,E2 -9788.743} C_VEL
LIN {X 0,Y 425.744,Z 299.844,A -85,B 0,C 180,E1 -9792.219,E2 -9792.219} C_VEL
LIN {X 0,Y 425.272,Z 314.536,A -85,B 0,C 180,E1 -9795.107,E2 -9795.107} C_VEL
LIN {X 0,Y 428.118,Z 338.401,A -85,B 0,C 180,E1 -9795.657,E2 -9795.657} C_VEL
LIN {X 0,Y 427.538,Z 393.79,A -85,B 0,C 180,E1 -9796.677,E2 -9796.677} C_VEL
LIN {X 0,Y 427.186,Z 405.161,A -85,B 0,C 180,E1 -9797.047,E2 -9797.047} C_VEL
LIN {X 0,Y 426.653,Z 416.639,A -85,B 0,C 180,E1 -9797.635,E2 -9797.635} C_VEL
LIN {X 0,Y 426.25,Z 425.301,A -85,B 0,C 180,E1 -9798.227,E2 -9798.227} C_VEL
LIN {X 0,Y 425.776,Z 433.617,A -85,B 0,C 180,E1 -9798.938,E2 -9798.938} C_VEL
LIN {X 0,Y 425.392,Z 441.522,A -85,B 0,C 180,E1 -9799.77,E2 -9799.77} C_VEL
LIN {X 0,Y 424.986,Z 448.935,A -85,B 0,C 180,E1 -9800.722,E2 -9800.722} C_VEL
LIN {X 0,Y 424.611,Z 456.468,A -85,B 0,C 180,E1 -9801.913,E2 -9801.913} C_VEL
LIN {X 0,Y 424.428,Z 462.38,A -85,B 0,C 180,E1 -9803.105,E2 -9803.105} C_VEL
LIN {X 0,Y 424.237,Z 467.057,A -85,B 0,C 180,E1 -9804.296,E2 -9804.296} C_VEL
LIN {X 0,Y 424.236,Z 470.106,A -85,B 0,C 180,E1 -9805.249,E2 -9805.249} C_VEL
LIN {X 0,Y 424.158,Z 472.49,A -85,B 0,C 180,E1 -9806.2,E2 -9806.2} C_VEL
LIN {X 0,Y 424.237,Z 474.258,A -85,B 0,C 180,E1 -9807.152,E2 -9807.152} C_VEL
LIN {X 0,Y 424.189,Z 475.507,A -85,B 0,C 180,E1 -9808.101,E2 -9808.101} C_VEL
LIN {X 0,Y 424.166,Z 476.268,A -85,B 0,C 180,E1 -9809.051,E2 -9809.051} C_VEL
LIN {X 0,Y 424.198,Z 476.555,A -85,B 0,C 180,E1 -9810,E2 -9810} C_VEL
LIN {X 0,Y 424.177,Z 476.258,A -85,B 0,C 180,E1 -9810.95,E2 -9810.95} C_VEL
LIN {X 0,Y 424.189,Z 475.409,A -85,B 0,C 180,E1 -9811.899,E2 -9811.899} C_VEL
LIN {X 0,Y 424.258,Z 474.071,A -85,B 0,C 180,E1 -9812.849,E2 -9812.849} C_VEL
LIN {X 0,Y 424.177,Z 471.04,A -85,B 0,C 180,E1 -9814.276,E2 -9814.276} C_VEL
LIN {X 0,Y 424.237,Z 466.702,A -85,B 0,C 180,E1 -9815.705,E2 -9815.705} C_VEL
LIN {X 0,Y 424.449,Z 460.666,A -85,B 0,C 180,E1 -9817.134,E2 -9817.134} C_VEL
LIN {X 0,Y 424.609,Z 455.654,A -85,B 0,C 180,E1 -9818.088,E2 -9818.088} C_VEL
LIN {X 0,Y 424.897,Z 449.614,A -85,B 0,C 180,E1 -9819.041,E2 -9819.041} C_VEL
LIN {X 0,Y 425.228,Z 442.257,A -85,B 0,C 180,E1 -9819.994,E2 -9819.994} C_VEL
LIN {X 0,Y 425.578,Z 434.391,A -85,B 0,C 180,E1 -9820.827,E2 -9820.827} C_VEL
LIN {X 0,Y 425.999,Z 426.111,A -85,B 0,C 180,E1 -9821.539,E2 -9821.539} C_VEL
LIN {X 0,Y 426.454,Z 415.604,A -85,B 0,C 180,E1 -9822.25,E2 -9822.25} C_VEL
LIN {X 0,Y 426.879,Z 404.454,A -85,B 0,C 180,E1 -9822.781,E2 -9822.781} C_VEL
LIN {X 0,Y 427.227,Z 394.227,A -85,B 0,C 180,E1 -9823.103,E2 -9823.103} C_VEL
LIN {X 0,Y 427.724,Z 338.181,A -85,B 0,C 180,E1 -9824.122,E2 -9824.122} C_VEL
LIN {X 0,Y 425.204,Z 315.787,A -85,B 0,C 180,E1 -9824.63,E2 -9824.63} C_VEL
LIN {X 0,Y 425.923,Z 298.069,A -85,B 0,C 180,E1 -9828.271,E2 -9828.271} C_VEL
LIN {X 0,Y 426.7,Z 282.525,A -85,B 0,C 180,E1 -9831.498,E2 -9831.498} C_VEL
LIN {X 0,Y 427.178,Z 272.913,A -85,B 0,C 180,E1 -9833.513,E2 -9833.513} C_VEL
LIN {X 0,Y 425.344,Z 262.318,A -85,B 0,C 180,E1 -9835.901,E2 -9835.901} C_VEL
LIN {X 0,Y 425.33,Z 262.315,A -85,B 0,C 180,E1 -9838.865,E2 -9838.865} C_VEL
LIN {X 0,Y 425.265,Z 262.323,A -85,B 0,C 180,E1 -9841.926,E2 -9841.926} C_VEL
LIN {X 0,Y 425.299,Z 262.321,A -85,B 0,C 180,E1 -9845.335,E2 -9845.335} C_VEL
LIN {X 0,Y 425.3,Z 262.318,A -85,B 0,C 180,E1 -9849.043,E2 -9849.043} C_VEL
LIN {X 0,Y 425.274,Z 262.319,A -85,B 0,C 180,E1 -9852.652,E2 -9852.652} C_VEL
LIN {X 0,Y 425.26,Z 262.323,A -85,B 0,C 180,E1 -9856.043,E2 -9856.043} C_VEL
LIN {X 0,Y 425.272,Z 262.32,A -85,B 0,C 180,E1 -9858.621,E2 -9858.621} C_VEL
LIN {X 0,Y 425.295,Z 262.319,A -85,B 0,C 180,E1 -9861.1,E2 -9861.1} C_VEL
LIN {X 0,Y 425.298,Z 262.316,A -85,B 0,C 180,E1 -9864.663,E2 -9864.663} C_VEL
LIN {X 0,Y 425.261,Z 262.323,A -85,B 0,C 180,E1 -9868.072,E2 -9868.072} C_VEL
LIN {X 0,Y 425.328,Z 262.318,A -85,B 0,C 180,E1 -9871.367,E2 -9871.367} C_VEL
LIN {X 0,Y 425.292,Z 262.317,A -85,B 0,C 180,E1 -9874.554,E2 -9874.554} C_VEL
LIN {X 0,Y 425.284,Z 262.324,A -85,B 0,C 180,E1 -9877.66,E2 -9877.66} C_VEL
LIN {X 0,Y 425.358,Z 262.309,A -85,B 0,C 180,E1 -9880.703,E2 -9880.703} C_VEL
LIN {X 0,Y 425.384,Z 262.312,A -85,B 0,C 180,E1 -9883.687,E2 -9883.687} C_VEL
LIN {X 0,Y 425.407,Z 262.31,A -85,B 0,C 180,E1 -9887.597,E2 -9887.597} C_VEL
LIN {X 0,Y 425.437,Z 262.305,A -85,B 0,C 180,E1 -9891.449,E2 -9891.449} C_VEL
LIN {X 0,Y 425.548,Z 262.286,A -85,B 0,C 180,E1 -9894.312,E2 -9894.312} C_VEL
LIN {X 0,Y 425.569,Z 262.284,A -85,B 0,C 180,E1 -9898.106,E2 -9898.106} C_VEL
LIN {X 0,Y 425.697,Z 262.269,A -85,B 0,C 180,E1 -9899.999,E2 -9899.999} C_VEL
LIN {X 0,Y 425.551,Z 262.286,A -85,B 0,C 180,E1 -9902.839,E2 -9902.839} C_VEL
LIN {X 0,Y 425.523,Z 262.289,A -85,B 0,C 180,E1 -9906.65,E2 -9906.65} C_VEL
LIN {X 0,Y 425.396,Z 262.31,A -85,B 0,C 180,E1 -9909.509,E2 -9909.509} C_VEL
LIN {X 0,Y 425.397,Z 262.305,A -85,B 0,C 180,E1 -9912.909,E2 -9912.909} C_VEL
LIN {X 0,Y 425.354,Z 262.31,A -85,B 0,C 180,E1 -9916.604,E2 -9916.604} C_VEL
LIN {X 0,Y 425.353,Z 262.317,A -85,B 0,C 180,E1 -9919.647,E2 -9919.647} C_VEL
LIN {X 0,Y 425.299,Z 262.321,A -85,B 0,C 180,E1 -9923.364,E2 -9923.364} C_VEL
LIN {X 0,Y 425.34,Z 262.312,A -85,B 0,C 180,E1 -9926.844,E2 -9926.844} C_VEL
LIN {X 0,Y 425.282,Z 262.325,A -85,B 0,C 180,E1 -9929.719,E2 -9929.719} C_VEL
LIN {X 0,Y 425.273,Z 262.321,A -85,B 0,C 180,E1 -9933.047,E2 -9933.047} C_VEL
LIN {X 0,Y 425.276,Z 262.323,A -85,B 0,C 180,E1 -9935.929,E2 -9935.929} C_VEL
LIN {X 0,Y 425.304,Z 262.317,A -85,B 0,C 180,E1 -9939.045,E2 -9939.045} C_VEL
LIN {X 0,Y 425.307,Z 262.319,A -85,B 0,C 180,E1 -9941.962,E2 -9941.962} C_VEL
LIN {X 0,Y 425.306,Z 262.319,A -85,B 0,C 180,E1 -9945.279,E2 -9945.279} C_VEL
LIN {X 0,Y 425.3,Z 262.317,A -85,B 0,C 180,E1 -9948.625,E2 -9948.625} C_VEL
LIN {X 0,Y 425.312,Z 262.317,A -85,B 0,C 180,E1 -9951.104,E2 -9951.104} C_VEL
LIN {X 0,Y 425.291,Z 262.318,A -85,B 0,C 180,E1 -9954.664,E2 -9954.664} C_VEL
LIN {X 0,Y 425.256,Z 262.325,A -85,B 0,C 180,E1 -9958.073,E2 -9958.073} C_VEL
LIN {X 0,Y 425.322,Z 262.317,A -85,B 0,C 180,E1 -9961.368,E2 -9961.368} C_VEL
LIN {X 0,Y 425.286,Z 262.319,A -85,B 0,C 180,E1 -9964.554,E2 -9964.554} C_VEL
LIN {X 0,Y 425.28,Z 262.326,A -85,B 0,C 180,E1 -9967.661,E2 -9967.661} C_VEL
LIN {X 0,Y 425.353,Z 262.311,A -85,B 0,C 180,E1 -9970.704,E2 -9970.704} C_VEL
LIN {X 0,Y 425.379,Z 262.314,A -85,B 0,C 180,E1 -9973.688,E2 -9973.688} C_VEL
LIN {X 0,Y 425.403,Z 262.31,A -85,B 0,C 180,E1 -9977.598,E2 -9977.598} C_VEL
LIN {X 0,Y 425.434,Z 262.304,A -85,B 0,C 180,E1 -9981.45,E2 -9981.45} C_VEL
LIN {X 0,Y 425.541,Z 262.288,A -85,B 0,C 180,E1 -9984.313,E2 -9984.313} C_VEL
LIN {X 0,Y 425.563,Z 262.286,A -85,B 0,C 180,E1 -9988.107,E2 -9988.107} C_VEL
LIN {X 0,Y 425.693,Z 262.271,A -85,B 0,C 180,E1 -9990,E2 -9990} C_VEL
LIN {X 0,Y 425.536,Z 262.288,A -85,B 0,C 180,E1 -9992.84,E2 -9992.84} C_VEL
LIN {X 0,Y 425.515,Z 262.291,A -85,B 0,C 180,E1 -9996.639,E2 -9996.639} C_VEL
LIN {X 0,Y 425.393,Z 262.307,A -85,B 0,C 180,E1 -9999.159,E2 -9999.159} C_VEL
LIN {X 0,Y 424.723,Z 262.394,A -85,B 0,C 180,E1 -9999.949,E2 -9999.949} C_VEL
LIN {X 0,Y 421.877,Z 262.745,A -85,B 0,C 180,E1 -10001.233,E2 -10001.233} C_VEL
LIN {X 0,Y 419.464,Z 263.045,A -85,B 0,C 180,E1 -10002.269,E2 -10002.269} C_VEL
LIN {X 0,Y 418.415,Z 263.176,A -85,B 0,C 180,E1 -10003.07,E2 -10003.07} C_VEL
LIN {X 0,Y 418.323,Z 263.189,A -85,B 0,C 180,E1 -10003.341,E2 -10003.341} C_VEL
LIN {X 0,Y 418.303,Z 263.189,A -85,B 0,C 180,E1 -10006.735,E2 -10006.735} C_VEL
LIN {X 0,Y 418.26,Z 263.2,A -85,B 0,C 180,E1 -10009.79,E2 -10009.79} C_VEL
LIN {X 0,Y 418.226,Z 263.199,A -85,B 0,C 180,E1 -10012.736,E2 -10012.736} C_VEL
LIN {X 0,Y 418.25,Z 263.2,A -85,B 0,C 180,E1 -10015.905,E2 -10015.905} C_VEL
LIN {X 0,Y 418.257,Z 263.195,A -85,B 0,C 180,E1 -10019.104,E2 -10019.104} C_VEL
LIN {X 0,Y 418.306,Z 263.314,A -85,B 0,C 180,E1 -10022.201,E2 -10022.201} C_VEL
LIN {X 0,Y 418.553,Z 268.743,A -85,B 0,C 180,E1 -10023.648,E2 -10023.648} C_VEL
LIN {X 0,Y 418.489,Z 271.074,A -85,B 0,C 180,E1 -10024.253,E2 -10024.253} C_VEL
LIN {X 0,Y 421.077,Z 285.158,A -85,B 0,C 180,E1 -10024.61,E2 -10024.61} C_VEL
LIN {X 0,Y 420.446,Z 347.818,A -85,B 0,C 180,E1 -10025.768,E2 -10025.768} C_VEL
LIN {X 0,Y 420.213,Z 358.839,A -85,B 0,C 180,E1 -10026.127,E2 -10026.127} C_VEL
LIN {X 0,Y 419.93,Z 370.75,A -85,B 0,C 180,E1 -10026.741,E2 -10026.741} C_VEL
LIN {X 0,Y 419.554,Z 380.006,A -85,B 0,C 180,E1 -10027.388,E2 -10027.388} C_VEL
LIN {X 0,Y 419.249,Z 388.515,A -85,B 0,C 180,E1 -10028.143,E2 -10028.143} C_VEL
LIN {X 0,Y 418.87,Z 396.279,A -85,B 0,C 180,E1 -10028.989,E2 -10028.989} C_VEL
LIN {X 0,Y 418.357,Z 404.825,A -85,B 0,C 180,E1 -10030.139,E2 -10030.139} C_VEL
